LIN {X 0,Y 446.477,Z 468.872,A -85,B 0,C 180,E1 -8659.303,E2 -8659.303} C_VEL
LIN {X 0,Y 446.426,Z 468.876,A -85,B 0,C 180,E1 -8662.2,E2 -8662.2} C_VEL
LIN {X 0,Y 446.445,Z 468.875,A -85,B 0,C 180,E1 -8665.153,E2 -8665.153} C_VEL
LIN {X 0,Y 446.494,Z 468.867,A -85,B 0,C 180,E1 -8668.178,E2 -8668.178} C_VEL
LIN {X 0,Y 446.427,Z 468.873,A -85,B 0,C 180,E1 -8671.774,E2 -8671.774} C_VEL
LIN {X 0,Y 446.437,Z 468.875,A -85,B 0,C 180,E1 -8674.523,E2 -8674.523} C_VEL
LIN {X 0,Y 446.423,Z 468.875,A -85,B 0,C 180,E1 -8678.079,E2 -8678.079} C_VEL
LIN {X 0,Y 446.435,Z 468.877,A -85,B 0,C 180,E1 -8680.917,E2 -8680.917} C_VEL
LIN {X 0,Y 446.408,Z 468.878,A -85,B 0,C 180,E1 -8683.846,E2 -8683.846} C_VEL
LIN {X 0,Y 446.406,Z 468.879,A -85,B 0,C 180,E1 -8686.403,E2 -8686.403} C_VEL
LIN {X 0,Y 446.435,Z 468.875,A -85,B 0,C 180,E1 -8689.082,E2 -8689.082} C_VEL
LIN {X 0,Y 446.412,Z 468.861,A -85,B 0,C 180,E1 -8692.12,E2 -8692.12} C_VEL
LIN {X 0,Y 446.428,Z 468.864,A -85,B 0,C 180,E1 -8695.475,E2 -8695.475} C_VEL
LIN {X 0,Y 446.475,Z 469.066,A -85,B 0,C 180,E1 -8698.572,E2 -8698.572} C_VEL
LIN {X 0,Y 449.548,Z 481.832,A -85,B 0,C 180,E1 -8700.754,E2 -8700.754} C_VEL
LIN {X 0,Y 450.889,Z 488.731,A -85,B 0,C 180,E1 -8701.866,E2 -8701.866} C_VEL
LIN {X 0,Y 450.438,Z 498.912,A -85,B 0,C 180,E1 -8703.346,E2 -8703.346} C_VEL
LIN {X 0,Y 449.183,Z 522.67,A -85,B 0,C 180,E1 -8706.728,E2 -8706.728} C_VEL
LIN {X 0,Y 447.86,Z 550.31,A -85,B 0,C 180,E1 -8710.583,E2 -8710.583} C_VEL
LIN {X 0,Y 447.484,Z 560.999,A -85,B 0,C 180,E1 -8712.017,E2 -8712.017} C_VEL
LIN {X 0,Y 450.722,Z 590.947,A -85,B 0,C 180,E1 -8712.672,E2 -8712.672} C_VEL
LIN {X 0,Y 449.9,Z 671.631,A -85,B 0,C 180,E1 -8713.988,E2 -8713.988} C_VEL
LIN {X 0,Y 449.488,Z 684.888,A -85,B 0,C 180,E1 -8714.38,E2 -8714.38} C_VEL
LIN {X 0,Y 448.906,Z 697.096,A -85,B 0,C 180,E1 -8714.912,E2 -8714.912} C_VEL
LIN {X 0,Y 448.274,Z 708.646,A -85,B 0,C 180,E1 -8715.587,E2 -8715.587} C_VEL
LIN {X 0,Y 447.599,Z 720.331,A -85,B 0,C 180,E1 -8716.472,E2 -8716.472} C_VEL
LIN {X 0,Y 447.145,Z 732.388,A -85,B 0,C 180,E1 -8717.518,E2 -8717.518} C_VEL
LIN {X 0,Y 446.594,Z 740.995,A -85,B 0,C 180,E1 -8718.424,E2 -8718.424} C_VEL
LIN {X 0,Y 446.277,Z 749.935,A -85,B 0,C 180,E1 -8719.565,E2 -8719.565} C_VEL
LIN {X 0,Y 445.963,Z 758.561,A -85,B 0,C 180,E1 -8720.931,E2 -8720.931} C_VEL
LIN {X 0,Y 445.725,Z 765.492,A -85,B 0,C 180,E1 -8722.296,E2 -8722.296} C_VEL
LIN {X 0,Y 445.62,Z 771.01,A -85,B 0,C 180,E1 -8723.66,E2 -8723.66} C_VEL
LIN {X 0,Y 445.591,Z 775.282,A -85,B 0,C 180,E1 -8725.022,E2 -8725.022} C_VEL
LIN {X 0,Y 445.584,Z 778.435,A -85,B 0,C 180,E1 -8726.381,E2 -8726.381} C_VEL
LIN {X 0,Y 445.572,Z 779.958,A -85,B 0,C 180,E1 -8727.286,E2 -8727.286} C_VEL
LIN {X 0,Y 445.593,Z 781.035,A -85,B 0,C 180,E1 -8728.191,E2 -8728.191} C_VEL
LIN {X 0,Y 445.531,Z 781.699,A -85,B 0,C 180,E1 -8729.095,E2 -8729.095} C_VEL
LIN {X 0,Y 445.555,Z 781.947,A -85,B 0,C 180,E1 -8729.998,E2 -8729.998} C_VEL
LIN {X 0,Y 445.528,Z 781.728,A -85,B 0,C 180,E1 -8730.902,E2 -8730.902} C_VEL
LIN {X 0,Y 445.589,Z 781.104,A -85,B 0,C 180,E1 -8731.806,E2 -8731.806} C_VEL
LIN {X 0,Y 445.567,Z 780.065,A -85,B 0,C 180,E1 -8732.711,E2 -8732.711} C_VEL
LIN {X 0,Y 445.573,Z 778.556,A -85,B 0,C 180,E1 -8733.616,E2 -8733.616} C_VEL
LIN {X 0,Y 445.578,Z 775.446,A -85,B 0,C 180,E1 -8734.975,E2 -8734.975} C_VEL
LIN {X 0,Y 445.604,Z 770.735,A -85,B 0,C 180,E1 -8736.47,E2 -8736.47} C_VEL
LIN {X 0,Y 445.745,Z 764.718,A -85,B 0,C 180,E1 -8737.928,E2 -8737.928} C_VEL
LIN {X 0,Y 445.979,Z 757.563,A -85,B 0,C 180,E1 -8739.294,E2 -8739.294} C_VEL
LIN {X 0,Y 446.321,Z 748.559,A -85,B 0,C 180,E1 -8740.661,E2 -8740.661} C_VEL
LIN {X 0,Y 446.658,Z 739.29,A -85,B 0,C 180,E1 -8741.802,E2 -8741.802} C_VEL
LIN {X 0,Y 447.233,Z 730.265,A -85,B 0,C 180,E1 -8742.707,E2 -8742.707} C_VEL
LIN {X 0,Y 447.641,Z 719.058,A -85,B 0,C 180,E1 -8743.619,E2 -8743.619} C_VEL
LIN {X 0,Y 448.409,Z 703.786,A -85,B 0,C 180,E1 -8744.637,E2 -8744.637} C_VEL
LIN {X 0,Y 448.973,Z 691.565,A -85,B 0,C 180,E1 -8745.257,E2 -8745.257} C_VEL
LIN {X 0,Y 449.538,Z 678.317,A -85,B 0,C 180,E1 -8745.731,E2 -8745.731} C_VEL
LIN {X 0,Y 449.81,Z 665.485,A -85,B 0,C 180,E1 -8746.012,E2 -8746.012} C_VEL
LIN {X 0,Y 450.296,Z 588.926,A -85,B 0,C 180,E1 -8747.238,E2 -8747.238} C_VEL
LIN {X 0,Y 447.405,Z 561.671,A -85,B 0,C 180,E1 -8747.804,E2 -8747.804} C_VEL
LIN {X 0,Y 448.284,Z 537.227,A -85,B 0,C 180,E1 -8751.134,E2 -8751.134} C_VEL
LIN {X 0,Y 449.315,Z 514.727,A -85,B 0,C 180,E1 -8754.24,E2 -8754.24} C_VEL
LIN {X 0,Y 450.483,Z 491.581,A -85,B 0,C 180,E1 -8757.481,E2 -8757.481} C_VEL
LIN {X 0,Y 450.402,Z 486.851,A -85,B 0,C 180,E1 -8758.163,E2 -8758.163} C_VEL
LIN {X 0,Y 446.49,Z 468.988,A -85,B 0,C 180,E1 -8760.996,E2 -8760.996} C_VEL
LIN {X 0,Y 446.416,Z 468.879,A -85,B 0,C 180,E1 -8764.522,E2 -8764.522} C_VEL
LIN {X 0,Y 446.392,Z 468.883,A -85,B 0,C 180,E1 -8768.075,E2 -8768.075} C_VEL
LIN {X 0,Y 446.398,Z 468.875,A -85,B 0,C 180,E1 -8771.392,E2 -8771.392} C_VEL
LIN {X 0,Y 446.441,Z 468.87,A -85,B 0,C 180,E1 -8775.102,E2 -8775.102} C_VEL
LIN {X 0,Y 446.401,Z 468.878,A -85,B 0,C 180,E1 -8778.605,E2 -8778.605} C_VEL
LIN {X 0,Y 446.4,Z 468.878,A -85,B 0,C 180,E1 -8781.92,E2 -8781.92} C_VEL
LIN {X 0,Y 446.417,Z 468.873,A -85,B 0,C 180,E1 -8785.476,E2 -8785.476} C_VEL
LIN {X 0,Y 446.404,Z 468.877,A -85,B 0,C 180,E1 -8788.698,E2 -8788.698} C_VEL
LIN {X 0,Y 446.473,Z 468.867,A -85,B 0,C 180,E1 -8791.82,E2 -8791.82} C_VEL
LIN {X 0,Y 446.426,Z 468.874,A -85,B 0,C 180,E1 -8794.845,E2 -8794.845} C_VEL
LIN {X 0,Y 446.435,Z 468.876,A -85,B 0,C 180,E1 -8798.244,E2 -8798.244} C_VEL
LIN {X 0,Y 446.442,Z 468.87,A -85,B 0,C 180,E1 -8801.648,E2 -8801.648} C_VEL
LIN {X 0,Y 446.493,Z 468.871,A -85,B 0,C 180,E1 -8804.479,E2 -8804.479} C_VEL
LIN {X 0,Y 446.505,Z 468.866,A -85,B 0,C 180,E1 -8808.192,E2 -8808.192} C_VEL
LIN {X 0,Y 446.586,Z 468.853,A -85,B 0,C 180,E1 -8811.857,E2 -8811.857} C_VEL
LIN {X 0,Y 446.624,Z 468.854,A -85,B 0,C 180,E1 -8814.582,E2 -8814.582} C_VEL
LIN {X 0,Y 446.651,Z 468.847,A -85,B 0,C 180,E1 -8818.196,E2 -8818.196} C_VEL
LIN {X 0,Y 446.778,Z 468.829,A -85,B 0,C 180,E1 -8820,E2 -8820} C_VEL
LIN {X 0,Y 446.694,Z 468.844,A -85,B 0,C 180,E1 -8822.705,E2 -8822.705} C_VEL
LIN {X 0,Y 446.624,Z 468.851,A -85,B 0,C 180,E1 -8826.324,E2 -8826.324} C_VEL
LIN {X 0,Y 446.525,Z 468.862,A -85,B 0,C 180,E1 -8829.055,E2 -8829.055} C_VEL
LIN {X 0,Y 446.507,Z 468.868,A -85,B 0,C 180,E1 -8832.73,E2 -8832.73} C_VEL
LIN {X 0,Y 446.482,Z 468.867,A -85,B 0,C 180,E1 -8836.228,E2 -8836.228} C_VEL
LIN {X 0,Y 446.455,Z 468.869,A -85,B 0,C 180,E1 -8839.303,E2 -8839.303} C_VEL
LIN {X 0,Y 446.404,Z 468.876,A -85,B 0,C 180,E1 -8842.2,E2 -8842.2} C_VEL
LIN {X 0,Y 446.444,Z 468.872,A -85,B 0,C 180,E1 -8845.153,E2 -8845.153} C_VEL
LIN {X 0,Y 446.471,Z 468.867,A -85,B 0,C 180,E1 -8848.179,E2 -8848.179} C_VEL
LIN {X 0,Y 446.406,Z 468.874,A -85,B 0,C 180,E1 -8851.776,E2 -8851.776} C_VEL
LIN {X 0,Y 446.417,Z 468.877,A -85,B 0,C 180,E1 -8854.524,E2 -8854.524} C_VEL
LIN {X 0,Y 446.418,Z 468.873,A -85,B 0,C 180,E1 -8858.083,E2 -8858.083} C_VEL
LIN {X 0,Y 446.416,Z 468.88,A -85,B 0,C 180,E1 -8860.919,E2 -8860.919} C_VEL
LIN {X 0,Y 446.414,Z 468.873,A -85,B 0,C 180,E1 -8863.844,E2 -8863.844} C_VEL
LIN {X 0,Y 446.436,Z 468.872,A -85,B 0,C 180,E1 -8866.398,E2 -8866.398} C_VEL
LIN {X 0,Y 446.459,Z 468.867,A -85,B 0,C 180,E1 -8869.806,E2 -8869.806} C_VEL
LIN {X 0,Y 446.424,Z 468.872,A -85,B 0,C 180,E1 -8872.125,E2 -8872.125} C_VEL
LIN {X 0,Y 446.421,Z 468.874,A -85,B 0,C 180,E1 -8875.478,E2 -8875.478} C_VEL
LIN {X 0,Y 446.408,Z 468.878,A -85,B 0,C 180,E1 -8878.701,E2 -8878.701} C_VEL
LIN {X 0,Y 446.476,Z 468.865,A -85,B 0,C 180,E1 -8881.823,E2 -8881.823} C_VEL
LIN {X 0,Y 446.451,Z 468.874,A -85,B 0,C 180,E1 -8884.849,E2 -8884.849} C_VEL
LIN {X 0,Y 446.442,Z 468.87,A -85,B 0,C 180,E1 -8888.246,E2 -8888.246} C_VEL
LIN {X 0,Y 446.452,Z 468.87,A -85,B 0,C 180,E1 -8891.651,E2 -8891.651} C_VEL
LIN {X 0,Y 446.503,Z 468.863,A -85,B 0,C 180,E1 -8894.481,E2 -8894.481} C_VEL
LIN {X 0,Y 446.514,Z 468.86,A -85,B 0,C 180,E1 -8898.195,E2 -8898.195} C_VEL
LIN {X 0,Y 446.597,Z 468.855,A -85,B 0,C 180,E1 -8901.859,E2 -8901.859} C_VEL
LIN {X 0,Y 446.645,Z 468.85,A -85,B 0,C 180,E1 -8904.584,E2 -8904.584} C_VEL
LIN {X 0,Y 446.462,Z 468.873,A -85,B 0,C 180,E1 -8905.655,E2 -8905.655} C_VEL
LIN {X 0,Y 446.343,Z 469.733,A -85,B 0,C 180,E1 -8906.036,E2 -8906.036} C_VEL
LIN {X 0,Y 446,Z 472.43,A -85,B 0,C 180,E1 -8906.43,E2 -8906.43} C_VEL
LIN {X 0,Y 445.49,Z 476.63,A -85,B 0,C 180,E1 -8906.744,E2 -8906.744} C_VEL
LIN {X 0,Y 444.895,Z 481.645,A -85,B 0,C 180,E1 -8906.929,E2 -8906.929} C_VEL
LIN {X 0,Y 444.052,Z 488.483,A -85,B 0,C 180,E1 -8907.053,E2 -8907.053} C_VEL
LIN {X 0,Y 443.816,Z 497.703,A -85,B 0,C 180,E1 -8907.197,E2 -8907.197} C_VEL
LIN {X 0,Y 443.446,Z 550.424,A -85,B 0,C 180,E1 -8908.072,E2 -8908.072} C_VEL
LIN {X 0,Y 443.362,Z 563.699,A -85,B 0,C 180,E1 -8908.469,E2 -8908.469} C_VEL
LIN {X 0,Y 443.164,Z 576.191,A -85,B 0,C 180,E1 -8909.029,E2 -8909.029} C_VEL
LIN {X 0,Y 442.841,Z 588.103,A -85,B 0,C 180,E1 -8909.752,E2 -8909.752} C_VEL
LIN {X 0,Y 442.363,Z 599.846,A -85,B 0,C 180,E1 -8910.684,E2 -8910.684} C_VEL
LIN {X 0,Y 441.805,Z 610.165,A -85,B 0,C 180,E1 -8911.711,E2 -8911.711} C_VEL
LIN {X 0,Y 441.426,Z 618.569,A -85,B 0,C 180,E1 -8912.739,E2 -8912.739} C_VEL
LIN {X 0,Y 440.972,Z 626.354,A -85,B 0,C 180,E1 -8913.885,E2 -8913.885} C_VEL
LIN {X 0,Y 440.548,Z 633.965,A -85,B 0,C 180,E1 -8915.265,E2 -8915.265} C_VEL
LIN {X 0,Y 440.134,Z 640.974,A -85,B 0,C 180,E1 -8916.88,E2 -8916.88} C_VEL
LIN {X 0,Y 439.824,Z 645.658,A -85,B 0,C 180,E1 -8918.27,E2 -8918.27} C_VEL
LIN {X 0,Y 439.587,Z 649.245,A -85,B 0,C 180,E1 -8919.666,E2 -8919.666} C_VEL
LIN {X 0,Y 439.392,Z 651.829,A -85,B 0,C 180,E1 -8921.067,E2 -8921.067} C_VEL
LIN {X 0,Y 439.334,Z 653.59,A -85,B 0,C 180,E1 -8922.629,E2 -8922.629} C_VEL
LIN {X 0,Y 439.316,Z 654.165,A -85,B 0,C 180,E1 -8923.886,E2 -8923.886} C_VEL
LIN {X 0,Y 439.329,Z 654.148,A -85,B 0,C 180,E1 -8924.832,E2 -8924.832} C_VEL
LIN {X 0,Y 439.453,Z 653.235,A -85,B 0,C 180,E1 -8926.352,E2 -8926.352} C_VEL
LIN {X 0,Y 439.592,Z 651.532,A -85,B 0,C 180,E1 -8927.685,E2 -8927.685} C_VEL
LIN {X 0,Y 439.838,Z 648.839,A -85,B 0,C 180,E1 -8929.076,E2 -8929.076} C_VEL
LIN {X 0,Y 440.172,Z 644.841,A -85,B 0,C 180,E1 -8930.566,E2 -8930.566} C_VEL
LIN {X 0,Y 440.575,Z 640.008,A -85,B 0,C 180,E1 -8931.938,E2 -8931.938} C_VEL
LIN {X 0,Y 441.03,Z 634.312,A -85,B 0,C 180,E1 -8933.23,E2 -8933.23} C_VEL
LIN {X 0,Y 441.595,Z 626.745,A -85,B 0,C 180,E1 -8934.612,E2 -8934.612} C_VEL
LIN {X 0,Y 442.19,Z 617.836,A -85,B 0,C 180,E1 -8935.919,E2 -8935.919} C_VEL
LIN {X 0,Y 442.747,Z 608.82,A -85,B 0,C 180,E1 -8936.995,E2 -8936.995} C_VEL
LIN {X 0,Y 443.35,Z 598.313,A -85,B 0,C 180,E1 -8938.011,E2 -8938.011} C_VEL
LIN {X 0,Y 443.885,Z 586.926,A -85,B 0,C 180,E1 -8938.877,E2 -8938.877} C_VEL
LIN {X 0,Y 444.236,Z 574.989,A -85,B 0,C 180,E1 -8939.581,E2 -8939.581} C_VEL
LIN {X 0,Y 444.407,Z 562.171,A -85,B 0,C 180,E1 -8940.133,E2 -8940.133} C_VEL
LIN {X 0,Y 444.504,Z 548.688,A -85,B 0,C 180,E1 -8940.496,E2 -8940.496} C_VEL
LIN {X 0,Y 445.006,Z 483.958,A -85,B 0,C 180,E1 -8941.582,E2 -8941.582} C_VEL
LIN {X 0,Y 439.597,Z 470.681,A -85,B 0,C 180,E1 -8942.108,E2 -8942.108} C_VEL
LIN {X 0,Y 439.42,Z 469.824,A -85,B 0,C 180,E1 -8942.299,E2 -8942.299} C_VEL
LIN {X 0,Y 439.395,Z 469.751,A -85,B 0,C 180,E1 -8945.341,E2 -8945.341} C_VEL
LIN {X 0,Y 439.379,Z 469.757,A -85,B 0,C 180,E1 -8948.597,E2 -8948.597} C_VEL
LIN {X 0,Y 439.393,Z 469.752,A -85,B 0,C 180,E1 -8951.258,E2 -8951.258} C_VEL
LIN {X 0,Y 439.404,Z 469.753,A -85,B 0,C 180,E1 -8954.731,E2 -8954.731} C_VEL
LIN {X 0,Y 439.401,Z 469.752,A -85,B 0,C 180,E1 -8957.797,E2 -8957.797} C_VEL
LIN {X 0,Y 439.449,Z 469.899,A -85,B 0,C 180,E1 -8960.531,E2 -8960.531} C_VEL
LIN {X 0,Y 442.432,Z 484.435,A -85,B 0,C 180,E1 -8963.155,E2 -8963.155} C_VEL
LIN {X 0,Y 441.997,Z 500.844,A -85,B 0,C 180,E1 -8965.883,E2 -8965.883} C_VEL
LIN {X 0,Y 441.36,Z 520.086,A -85,B 0,C 180,E1 -8969.045,E2 -8969.045} C_VEL
LIN {X 0,Y 442.817,Z 528.551,A -85,B 0,C 180,E1 -8969.296,E2 -8969.296} C_VEL
LIN {X 0,Y 444.048,Z 537.306,A -85,B 0,C 180,E1 -8969.507,E2 -8969.507} C_VEL
LIN {X 0,Y 442.745,Z 630.209,A -85,B 0,C 180,E1 -8971.187,E2 -8971.187} C_VEL
LIN {X 0,Y 442.439,Z 643.262,A -85,B 0,C 180,E1 -8971.605,E2 -8971.605} C_VEL
LIN {X 0,Y 441.965,Z 656.195,A -85,B 0,C 180,E1 -8972.218,E2 -8972.218} C_VEL
LIN {X 0,Y 441.538,Z 668.066,A -85,B 0,C 180,E1 -8972.97,E2 -8972.97} C_VEL
LIN {X 0,Y 440.979,Z 679.22,A -85,B 0,C 180,E1 -8973.879,E2 -8973.879} C_VEL
LIN {X 0,Y 440.37,Z 690.05,A -85,B 0,C 180,E1 -8974.981,E2 -8974.981} C_VEL
LIN {X 0,Y 439.881,Z 699.698,A -85,B 0,C 180,E1 -8976.208,E2 -8976.208} C_VEL
LIN {X 0,Y 439.385,Z 708.731,A -85,B 0,C 180,E1 -8977.635,E2 -8977.635} C_VEL
LIN {X 0,Y 438.971,Z 716.196,A -85,B 0,C 180,E1 -8979.132,E2 -8979.132} C_VEL
LIN {X 0,Y 438.729,Z 722.312,A -85,B 0,C 180,E1 -8980.705,E2 -8980.705} C_VEL
LIN {X 0,Y 438.498,Z 726.876,A -85,B 0,C 180,E1 -8982.271,E2 -8982.271} C_VEL
LIN {X 0,Y 438.419,Z 728.978,A -85,B 0,C 180,E1 -8983.229,E2 -8983.229} C_VEL
LIN {X 0,Y 438.327,Z 730.625,A -85,B 0,C 180,E1 -8984.183,E2 -8984.183} C_VEL
LIN {X 0,Y 438.293,Z 731.781,A -85,B 0,C 180,E1 -8985.134,E2 -8985.134} C_VEL
LIN {X 0,Y 438.252,Z 732.499,A -85,B 0,C 180,E1 -8986.082,E2 -8986.082} C_VEL
LIN {X 0,Y 438.272,Z 732.802,A -85,B 0,C 180,E1 -8987.027,E2 -8987.027} C_VEL
LIN {X 0,Y 438.381,Z 732.633,A -85,B 0,C 180,E1 -8987.971,E2 -8987.971} C_VEL
LIN {X 0,Y 438.381,Z 732.047,A -85,B 0,C 180,E1 -8988.909,E2 -8988.909} C_VEL
LIN {X 0,Y 438.369,Z 731.061,A -85,B 0,C 180,E1 -8989.843,E2 -8989.843} C_VEL
LIN {X 0,Y 438.443,Z 729.611,A -85,B 0,C 180,E1 -8990.776,E2 -8990.776} C_VEL
LIN {X 0,Y 438.654,Z 726.595,A -85,B 0,C 180,E1 -8992.173,E2 -8992.173} C_VEL
LIN {X 0,Y 438.836,Z 722.512,A -85,B 0,C 180,E1 -8993.564,E2 -8993.564} C_VEL
LIN {X 0,Y 439.121,Z 716.276,A -85,B 0,C 180,E1 -8995.18,E2 -8995.18} C_VEL
LIN {X 0,Y 439.472,Z 709.438,A -85,B 0,C 180,E1 -8996.562,E2 -8996.562} C_VEL
LIN {X 0,Y 440.004,Z 700.882,A -85,B 0,C 180,E1 -8997.941,E2 -8997.941} C_VEL
LIN {X 0,Y 440.58,Z 691.174,A -85,B 0,C 180,E1 -8999.201,E2 -8999.201} C_VEL
LIN {X 0,Y 441.227,Z 680.069,A -85,B 0,C 180,E1 -9000.343,E2 -9000.343} C_VEL
LIN {X 0,Y 441.8,Z 668.964,A -85,B 0,C 180,E1 -9001.254,E2 -9001.254} C_VEL
LIN {X 0,Y 442.291,Z 657.378,A -85,B 0,C 180,E1 -9001.992,E2 -9001.992} C_VEL
LIN {X 0,Y 442.762,Z 644.338,A -85,B 0,C 180,E1 -9002.616,E2 -9002.616} C_VEL
LIN {X 0,Y 443.053,Z 631.125,A -85,B 0,C 180,E1 -9003.041,E2 -9003.041} C_VEL
LIN {X 0,Y 444.582,Z 535.636,A -85,B 0,C 180,E1 -9004.853,E2 -9004.853} C_VEL
LIN {X 0,Y 442.01,Z 521.914,A -85,B 0,C 180,E1 -9005.295,E2 -9005.295} C_VEL
LIN {X 0,Y 442.645,Z 499.692,A -85,B 0,C 180,E1 -9008.906,E2 -9008.906} C_VEL
LIN {X 0,Y 443.011,Z 486.705,A -85,B 0,C 180,E1 -9010.975,E2 -9010.975} C_VEL
LIN {X 0,Y 441.276,Z 477.085,A -85,B 0,C 180,E1 -9012.65,E2 -9012.65} C_VEL
LIN {X 0,Y 439.441,Z 469.873,A -85,B 0,C 180,E1 -9013.969,E2 -9013.969} C_VEL
LIN {X 0,Y 439.456,Z 469.747,A -85,B 0,C 180,E1 -9016.731,E2 -9016.731} C_VEL
LIN {X 0,Y 439.41,Z 469.751,A -85,B 0,C 180,E1 -9019.626,E2 -9019.626} C_VEL
LIN {X 0,Y 439.372,Z 469.756,A -85,B 0,C 180,E1 -9022.575,E2 -9022.575} C_VEL
LIN {X 0,Y 439.394,Z 469.752,A -85,B 0,C 180,E1 -9025.586,E2 -9025.586} C_VEL
LIN {X 0,Y 439.426,Z 469.749,A -85,B 0,C 180,E1 -9028.673,E2 -9028.673} C_VEL
LIN {X 0,Y 439.378,Z 469.752,A -85,B 0,C 180,E1 -9032.03,E2 -9032.03} C_VEL
LIN {X 0,Y 439.403,Z 469.749,A -85,B 0,C 180,E1 -9035.34,E2 -9035.34} C_VEL
LIN {X 0,Y 439.386,Z 469.754,A -85,B 0,C 180,E1 -9038.595,E2 -9038.595} C_VEL
LIN {X 0,Y 439.397,Z 469.751,A -85,B 0,C 180,E1 -9041.256,E2 -9041.256} C_VEL
LIN {X 0,Y 439.408,Z 469.751,A -85,B 0,C 180,E1 -9044.729,E2 -9044.729} C_VEL
LIN {X 0,Y 439.404,Z 469.751,A -85,B 0,C 180,E1 -9047.795,E2 -9047.795} C_VEL
LIN {X 0,Y 439.397,Z 469.747,A -85,B 0,C 180,E1 -9050.223,E2 -9050.223} C_VEL
LIN {X 0,Y 439.379,Z 469.754,A -85,B 0,C 180,E1 -9053.712,E2 -9053.712} C_VEL
LIN {X 0,Y 439.378,Z 469.754,A -85,B 0,C 180,E1 -9057.053,E2 -9057.053} C_VEL
LIN {X 0,Y 439.408,Z 469.966,A -85,B 0,C 180,E1 -9058.242,E2 -9058.242} C_VEL
LIN {X 0,Y 442.211,Z 481.198,A -85,B 0,C 180,E1 -9060.22,E2 -9060.22} C_VEL
LIN {X 0,Y 443.966,Z 489.822,A -85,B 0,C 180,E1 -9061.646,E2 -9061.646} C_VEL
LIN {X 0,Y 444.057,Z 493.291,A -85,B 0,C 180,E1 -9062.178,E2 -9062.178} C_VEL
LIN {X 0,Y 442.567,Z 516.885,A -85,B 0,C 180,E1 -9065.613,E2 -9065.613} C_VEL
LIN {X 0,Y 441.379,Z 538.889,A -85,B 0,C 180,E1 -9068.761,E2 -9068.761} C_VEL
LIN {X 0,Y 440.535,Z 559.742,A -85,B 0,C 180,E1 -9071.674,E2 -9071.674} C_VEL
LIN {X 0,Y 443.258,Z 584.816,A -85,B 0,C 180,E1 -9072.251,E2 -9072.251} C_VEL
LIN {X 0,Y 443.978,Z 592.474,A -85,B 0,C 180,E1 -9072.412,E2 -9072.412} C_VEL
LIN {X 0,Y 443.12,Z 670.409,A -85,B 0,C 180,E1 -9073.707,E2 -9073.707} C_VEL
LIN {X 0,Y 442.711,Z 683.725,A -85,B 0,C 180,E1 -9074.106,E2 -9074.106} C_VEL
LIN {X 0,Y 442.024,Z 696.533,A -85,B 0,C 180,E1 -9074.671,E2 -9074.671} C_VEL
LIN {X 0,Y 441.371,Z 707.968,A -85,B 0,C 180,E1 -9075.357,E2 -9075.357} C_VEL
LIN {X 0,Y 440.365,Z 725.352,A -85,B 0,C 180,E1 -9076.701,E2 -9076.701} C_VEL
LIN {X 0,Y 439.949,Z 735.393,A -85,B 0,C 180,E1 -9077.662,E2 -9077.662} C_VEL
LIN {X 0,Y 439.51,Z 744.355,A -85,B 0,C 180,E1 -9078.702,E2 -9078.702} C_VEL
LIN {X 0,Y 439.078,Z 752.595,A -85,B 0,C 180,E1 -9079.858,E2 -9079.858} C_VEL
LIN {X 0,Y 438.812,Z 760.649,A -85,B 0,C 180,E1 -9081.247,E2 -9081.247} C_VEL
LIN {X 0,Y 438.614,Z 767.072,A -85,B 0,C 180,E1 -9082.634,E2 -9082.634} C_VEL
LIN {X 0,Y 438.496,Z 772.591,A -85,B 0,C 180,E1 -9084.154,E2 -9084.154} C_VEL
LIN {X 0,Y 438.47,Z 776.04,A -85,B 0,C 180,E1 -9085.402,E2 -9085.402} C_VEL
LIN {X 0,Y 438.48,Z 778.049,A -85,B 0,C 180,E1 -9086.323,E2 -9086.323} C_VEL
LIN {X 0,Y 438.495,Z 779.568,A -85,B 0,C 180,E1 -9087.242,E2 -9087.242} C_VEL
LIN {X 0,Y 438.5,Z 780.643,A -85,B 0,C 180,E1 -9088.162,E2 -9088.162} C_VEL
LIN {X 0,Y 438.465,Z 781.308,A -85,B 0,C 180,E1 -9089.08,E2 -9089.08} C_VEL
LIN {X 0,Y 438.484,Z 781.546,A -85,B 0,C 180,E1 -9089.998,E2 -9089.998} C_VEL
LIN {X 0,Y 438.462,Z 781.32,A -85,B 0,C 180,E1 -9090.917,E2 -9090.917} C_VEL
LIN {X 0,Y 438.496,Z 780.688,A -85,B 0,C 180,E1 -9091.835,E2 -9091.835} C_VEL
LIN {X 0,Y 438.489,Z 779.642,A -85,B 0,C 180,E1 -9092.754,E2 -9092.754} C_VEL
LIN {X 0,Y 438.472,Z 778.114,A -85,B 0,C 180,E1 -9093.674,E2 -9093.674} C_VEL
LIN {X 0,Y 438.507,Z 774.981,A -85,B 0,C 180,E1 -9095.056,E2 -9095.056} C_VEL
LIN {X 0,Y 438.505,Z 770.719,A -85,B 0,C 180,E1 -9096.44,E2 -9096.44} C_VEL
LIN {X 0,Y 438.688,Z 764.185,A -85,B 0,C 180,E1 -9098.057,E2 -9098.057} C_VEL
LIN {X 0,Y 438.911,Z 756.97,A -85,B 0,C 180,E1 -9099.445,E2 -9099.445} C_VEL
LIN {X 0,Y 439.31,Z 747.921,A -85,B 0,C 180,E1 -9100.833,E2 -9100.833} C_VEL
LIN {X 0,Y 439.641,Z 738.578,A -85,B 0,C 180,E1 -9101.993,E2 -9101.993} C_VEL
LIN {X 0,Y 440.218,Z 729.467,A -85,B 0,C 180,E1 -9102.913,E2 -9102.913} C_VEL
LIN {X 0,Y 440.662,Z 718.157,A -85,B 0,C 180,E1 -9103.839,E2 -9103.839} C_VEL
LIN {X 0,Y 441.63,Z 700.367,A -85,B 0,C 180,E1 -9104.985,E2 -9104.985} C_VEL
LIN {X 0,Y 442.234,Z 687.379,A -85,B 0,C 180,E1 -9105.613,E2 -9105.613} C_VEL
LIN {X 0,Y 442.72,Z 674.287,A -85,B 0,C 180,E1 -9106.039,E2 -9106.039} C_VEL
LIN {X 0,Y 443.012,Z 655.783,A -85,B 0,C 180,E1 -9106.383,E2 -9106.383} C_VEL
LIN {X 0,Y 443.553,Z 590.85,A -85,B 0,C 180,E1 -9107.436,E2 -9107.436} C_VEL
LIN {X 0,Y 440.399,Z 560.897,A -85,B 0,C 180,E1 -9108.056,E2 -9108.056} C_VEL
LIN {X 0,Y 441.264,Z 537.756,A -85,B 0,C 180,E1 -9111.242,E2 -9111.242} C_VEL
LIN {X 0,Y 442.442,Z 513.843,A -85,B 0,C 180,E1 -9114.604,E2 -9114.604} C_VEL
LIN {X 0,Y 443.65,Z 490.977,A -85,B 0,C 180,E1 -9117.858,E2 -9117.858} C_VEL
LIN {X 0,Y 443.017,Z 486.063,A -85,B 0,C 180,E1 -9118.604,E2 -9118.604} C_VEL
LIN {X 0,Y 439.427,Z 469.862,A -85,B 0,C 180,E1 -9121.232,E2 -9121.232} C_VEL
LIN {X 0,Y 439.378,Z 469.758,A -85,B 0,C 180,E1 -9124.042,E2 -9124.042} C_VEL
LIN {X 0,Y 439.333,Z 469.756,A -85,B 0,C 180,E1 -9126.884,E2 -9126.884} C_VEL
LIN {X 0,Y 439.337,Z 469.758,A -85,B 0,C 180,E1 -9129.839,E2 -9129.839} C_VEL
LIN {X 0,Y 439.335,Z 469.758,A -85,B 0,C 180,E1 -9132.62,E2 -9132.62} C_VEL
LIN {X 0,Y 439.39,Z 469.748,A -85,B 0,C 180,E1 -9135.269,E2 -9135.269} C_VEL
LIN {X 0,Y 439.361,Z 469.754,A -85,B 0,C 180,E1 -9138.745,E2 -9138.745} C_VEL
LIN {X 0,Y 439.354,Z 469.753,A -85,B 0,C 180,E1 -9141.608,E2 -9141.608} C_VEL
LIN {X 0,Y 439.387,Z 469.75,A -85,B 0,C 180,E1 -9144.843,E2 -9144.843} C_VEL
LIN {X 0,Y 439.361,Z 469.757,A -85,B 0,C 180,E1 -9148.138,E2 -9148.138} C_VEL
LIN {X 0,Y 439.421,Z 469.745,A -85,B 0,C 180,E1 -9151.597,E2 -9151.597} C_VEL
LIN {X 0,Y 439.375,Z 469.757,A -85,B 0,C 180,E1 -9154.413,E2 -9154.413} C_VEL
LIN {X 0,Y 439.35,Z 469.753,A -85,B 0,C 180,E1 -9157.423,E2 -9157.423} C_VEL
LIN {X 0,Y 439.428,Z 469.748,A -85,B 0,C 180,E1 -9160.662,E2 -9160.662} C_VEL
LIN {X 0,Y 439.448,Z 469.746,A -85,B 0,C 180,E1 -9164.224,E2 -9164.224} C_VEL
LIN {X 0,Y 439.471,Z 469.74,A -85,B 0,C 180,E1 -9168.001,E2 -9168.001} C_VEL
LIN {X 0,Y 439.534,Z 469.73,A -85,B 0,C 180,E1 -9171.726,E2 -9171.726} C_VEL
LIN {X 0,Y 439.6,Z 469.73,A -85,B 0,C 180,E1 -9174.495,E2 -9174.495} C_VEL
LIN {X 0,Y 439.621,Z 469.722,A -85,B 0,C 180,E1 -9178.167,E2 -9178.167} C_VEL
LIN {X 0,Y 439.748,Z 469.705,A -85,B 0,C 180,E1 -9180,E2 -9180} C_VEL
LIN {X 0,Y 439.64,Z 469.722,A -85,B 0,C 180,E1 -9182.748,E2 -9182.748} C_VEL
LIN {X 0,Y 439.599,Z 469.728,A -85,B 0,C 180,E1 -9186.425,E2 -9186.425} C_VEL
LIN {X 0,Y 439.487,Z 469.737,A -85,B 0,C 180,E1 -9189.202,E2 -9189.202} C_VEL
LIN {X 0,Y 439.451,Z 469.744,A -85,B 0,C 180,E1 -9192.938,E2 -9192.938} C_VEL
LIN {X 0,Y 439.433,Z 469.746,A -85,B 0,C 180,E1 -9196.349,E2 -9196.349} C_VEL
LIN {X 0,Y 439.388,Z 469.748,A -85,B 0,C 180,E1 -9199.627,E2 -9199.627} C_VEL
LIN {X 0,Y 439.351,Z 469.759,A -85,B 0,C 180,E1 -9202.576,E2 -9202.576} C_VEL
LIN {X 0,Y 439.391,Z 469.748,A -85,B 0,C 180,E1 -9205.585,E2 -9205.585} C_VEL
LIN {X 0,Y 439.404,Z 469.753,A -85,B 0,C 180,E1 -9208.674,E2 -9208.674} C_VEL
LIN {X 0,Y 439.357,Z 469.752,A -85,B 0,C 180,E1 -9212.031,E2 -9212.031} C_VEL
LIN {X 0,Y 439.383,Z 469.751,A -85,B 0,C 180,E1 -9215.342,E2 -9215.342} C_VEL
LIN {X 0,Y 439.371,Z 469.755,A -85,B 0,C 180,E1 -9218.596,E2 -9218.596} C_VEL
LIN {X 0,Y 439.377,Z 469.752,A -85,B 0,C 180,E1 -9221.258,E2 -9221.258} C_VEL
LIN {X 0,Y 439.396,Z 469.753,A -85,B 0,C 180,E1 -9224.729,E2 -9224.729} C_VEL
LIN {X 0,Y 439.402,Z 469.746,A -85,B 0,C 180,E1 -9227.799,E2 -9227.799} C_VEL
LIN {X 0,Y 439.442,Z 469.742,A -85,B 0,C 180,E1 -9230.231,E2 -9230.231} C_VEL
LIN {X 0,Y 439.367,Z 469.751,A -85,B 0,C 180,E1 -9233.714,E2 -9233.714} C_VEL
LIN {X 0,Y 439.364,Z 469.758,A -85,B 0,C 180,E1 -9237.055,E2 -9237.055} C_VEL
LIN {X 0,Y 439.374,Z 469.75,A -85,B 0,C 180,E1 -9240.276,E2 -9240.276} C_VEL
LIN {X 0,Y 439.422,Z 469.747,A -85,B 0,C 180,E1 -9243.398,E2 -9243.398} C_VEL
LIN {X 0,Y 439.38,Z 469.75,A -85,B 0,C 180,E1 -9246.431,E2 -9246.431} C_VEL
LIN {X 0,Y 439.383,Z 469.752,A -85,B 0,C 180,E1 -9249.399,E2 -9249.399} C_VEL
LIN {X 0,Y 439.426,Z 469.744,A -85,B 0,C 180,E1 -9252.311,E2 -9252.311} C_VEL
LIN {X 0,Y 439.443,Z 469.749,A -85,B 0,C 180,E1 -9255.176,E2 -9255.176} C_VEL
LIN {X 0,Y 439.48,Z 469.737,A -85,B 0,C 180,E1 -9258.003,E2 -9258.003} C_VEL
LIN {X 0,Y 439.545,Z 469.734,A -85,B 0,C 180,E1 -9261.728,E2 -9261.728} C_VEL
LIN {X 0,Y 439.621,Z 469.725,A -85,B 0,C 180,E1 -9264.497,E2 -9264.497} C_VEL
LIN {X 0,Y 439.477,Z 469.927,A -85,B 0,C 180,E1 -9266.438,E2 -9266.438} C_VEL
LIN {X 0,Y 439.764,Z 471.003,A -85,B 0,C 180,E1 -9266.592,E2 -9266.592} C_VEL
LIN {X 0,Y 443.948,Z 482.631,A -85,B 0,C 180,E1 -9266.953,E2 -9266.953} C_VEL
LIN {X 0,Y 443.816,Z 497.703,A -85,B 0,C 180,E1 -9267.197,E2 -9267.197} C_VEL
LIN {X 0,Y 443.12,Z 503.549,A -85,B 0,C 180,E1 -9267.269,E2 -9267.269} C_VEL
LIN {X 0,Y 437.287,Z 522.517,A -85,B 0,C 180,E1 -9267.377,E2 -9267.377} C_VEL
LIN {X 0,Y 436.633,Z 528.362,A -85,B 0,C 180,E1 -9267.452,E2 -9267.452} C_VEL
LIN {X 0,Y 436.576,Z 553.241,A -85,B 0,C 180,E1 -9267.897,E2 -9267.897} C_VEL
LIN {X 0,Y 436.478,Z 566.473,A -85,B 0,C 180,E1 -9268.325,E2 -9268.325} C_VEL
LIN {X 0,Y 436.264,Z 578.709,A -85,B 0,C 180,E1 -9268.905,E2 -9268.905} C_VEL
LIN {X 0,Y 435.94,Z 589.882,A -85,B 0,C 180,E1 -9269.618,E2 -9269.618} C_VEL
LIN {X 0,Y 435.455,Z 601.621,A -85,B 0,C 180,E1 -9270.58,E2 -9270.58} C_VEL
LIN {X 0,Y 434.873,Z 611.805,A -85,B 0,C 180,E1 -9271.622,E2 -9271.622} C_VEL
LIN {X 0,Y 434.432,Z 620.921,A -85,B 0,C 180,E1 -9272.783,E2 -9272.783} C_VEL
LIN {X 0,Y 433.84,Z 629.806,A -85,B 0,C 180,E1 -9274.182,E2 -9274.182} C_VEL
LIN {X 0,Y 433.427,Z 636.955,A -85,B 0,C 180,E1 -9275.585,E2 -9275.585} C_VEL
LIN {X 0,Y 433.114,Z 642.677,A -85,B 0,C 180,E1 -9276.992,E2 -9276.992} C_VEL
LIN {X 0,Y 432.769,Z 647.209,A -85,B 0,C 180,E1 -9278.406,E2 -9278.406} C_VEL
LIN {X 0,Y 432.598,Z 649.598,A -85,B 0,C 180,E1 -9279.351,E2 -9279.351} C_VEL
LIN {X 0,Y 432.474,Z 651.558,A -85,B 0,C 180,E1 -9280.299,E2 -9280.299} C_VEL
LIN {X 0,Y 432.35,Z 653.111,A -85,B 0,C 180,E1 -9281.25,E2 -9281.25} C_VEL
LIN {X 0,Y 432.329,Z 654.656,A -85,B 0,C 180,E1 -9282.745,E2 -9282.745} C_VEL
LIN {X 0,Y 432.299,Z 655.192,A -85,B 0,C 180,E1 -9284.116,E2 -9284.116} C_VEL
LIN {X 0,Y 432.337,Z 655.081,A -85,B 0,C 180,E1 -9285.077,E2 -9285.077} C_VEL
LIN {X 0,Y 432.459,Z 654.156,A -85,B 0,C 180,E1 -9286.5,E2 -9286.5} C_VEL
LIN {X 0,Y 432.623,Z 652.222,A -85,B 0,C 180,E1 -9287.98,E2 -9287.98} C_VEL
LIN {X 0,Y 432.952,Z 648.636,A -85,B 0,C 180,E1 -9289.696,E2 -9289.696} C_VEL
LIN {X 0,Y 433.405,Z 643.579,A -85,B 0,C 180,E1 -9291.4,E2 -9291.4} C_VEL
LIN {X 0,Y 433.881,Z 637.791,A -85,B 0,C 180,E1 -9292.878,E2 -9292.878} C_VEL
LIN {X 0,Y 434.53,Z 630.38,A -85,B 0,C 180,E1 -9294.359,E2 -9294.359} C_VEL
LIN {X 0,Y 435.12,Z 622.41,A -85,B 0,C 180,E1 -9295.647,E2 -9295.647} C_VEL
LIN {X 0,Y 435.821,Z 613.295,A -85,B 0,C 180,E1 -9296.843,E2 -9296.843} C_VEL
LIN {X 0,Y 436.334,Z 603.926,A -85,B 0,C 180,E1 -9297.848,E2 -9297.848} C_VEL
LIN {X 0,Y 436.987,Z 592.133,A -85,B 0,C 180,E1 -9298.849,E2 -9298.849} C_VEL
LIN {X 0,Y 437.41,Z 581.062,A -85,B 0,C 180,E1 -9299.588,E2 -9299.588} C_VEL
LIN {X 0,Y 437.69,Z 568.474,A -85,B 0,C 180,E1 -9300.219,E2 -9300.219} C_VEL
LIN {X 0,Y 437.809,Z 556.155,A -85,B 0,C 180,E1 -9300.643,E2 -9300.643} C_VEL
LIN {X 0,Y 437.835,Z 537.38,A -85,B 0,C 180,E1 -9301.015,E2 -9301.015} C_VEL
LIN {X 0,Y 438.401,Z 485.702,A -85,B 0,C 180,E1 -9301.882,E2 -9301.882} C_VEL
LIN {X 0,Y 432.634,Z 471.813,A -85,B 0,C 180,E1 -9302.445,E2 -9302.445} C_VEL
LIN {X 0,Y 432.407,Z 470.938,A -85,B 0,C 180,E1 -9302.561,E2 -9302.561} C_VEL
LIN {X 0,Y 432.354,Z 470.629,A -85,B 0,C 180,E1 -9302.995,E2 -9302.995} C_VEL
LIN {X 0,Y 432.34,Z 470.631,A -85,B 0,C 180,E1 -9305.819,E2 -9305.819} C_VEL
LIN {X 0,Y 432.331,Z 470.627,A -85,B 0,C 180,E1 -9309.346,E2 -9309.346} C_VEL
LIN {X 0,Y 432.337,Z 470.628,A -85,B 0,C 180,E1 -9311.798,E2 -9311.798} C_VEL
LIN {X 0,Y 432.338,Z 470.632,A -85,B 0,C 180,E1 -9314.348,E2 -9314.348} C_VEL
LIN {X 0,Y 432.325,Z 470.635,A -85,B 0,C 180,E1 -9317.017,E2 -9317.017} C_VEL
LIN {X 0,Y 432.439,Z 470.805,A -85,B 0,C 180,E1 -9320.306,E2 -9320.306} C_VEL
LIN {X 0,Y 435.55,Z 485.948,A -85,B 0,C 180,E1 -9323.054,E2 -9323.054} C_VEL
LIN {X 0,Y 435.058,Z 502.665,A -85,B 0,C 180,E1 -9325.851,E2 -9325.851} C_VEL
LIN {X 0,Y 434.461,Z 520.598,A -85,B 0,C 180,E1 -9328.8,E2 -9328.8} C_VEL
LIN {X 0,Y 437.236,Z 537.224,A -85,B 0,C 180,E1 -9329.244,E2 -9329.244} C_VEL
LIN {X 0,Y 435.889,Z 630.079,A -85,B 0,C 180,E1 -9330.958,E2 -9330.958} C_VEL
LIN {X 0,Y 435.563,Z 643.223,A -85,B 0,C 180,E1 -9331.379,E2 -9331.379} C_VEL
LIN {X 0,Y 435.05,Z 656.231,A -85,B 0,C 180,E1 -9331.999,E2 -9331.999} C_VEL
LIN {X 0,Y 434.594,Z 668.718,A -85,B 0,C 180,E1 -9332.804,E2 -9332.804} C_VEL
LIN {X 0,Y 433.954,Z 680.73,A -85,B 0,C 180,E1 -9333.812,E2 -9333.812} C_VEL
LIN {X 0,Y 433.331,Z 691.347,A -85,B 0,C 180,E1 -9334.931,E2 -9334.931} C_VEL
LIN {X 0,Y 432.88,Z 699.962,A -85,B 0,C 180,E1 -9336.054,E2 -9336.054} C_VEL
LIN {X 0,Y 432.419,Z 707.97,A -85,B 0,C 180,E1 -9337.32,E2 -9337.32} C_VEL
LIN {X 0,Y 432.007,Z 715.45,A -85,B 0,C 180,E1 -9338.779,E2 -9338.779} C_VEL
LIN {X 0,Y 431.737,Z 720.515,A -85,B 0,C 180,E1 -9340.011,E2 -9340.011} C_VEL
LIN {X 0,Y 431.53,Z 725.325,A -85,B 0,C 180,E1 -9341.484,E2 -9341.484} C_VEL
LIN {X 0,Y 431.373,Z 728.884,A -85,B 0,C 180,E1 -9342.947,E2 -9342.947} C_VEL
LIN {X 0,Y 431.247,Z 730.854,A -85,B 0,C 180,E1 -9344.057,E2 -9344.057} C_VEL
LIN {X 0,Y 431.218,Z 731.939,A -85,B 0,C 180,E1 -9344.885,E2 -9344.885} C_VEL
LIN {X 0,Y 431.165,Z 732.762,A -85,B 0,C 180,E1 -9345.848,E2 -9345.848} C_VEL
LIN {X 0,Y 431.19,Z 733.152,A -85,B 0,C 180,E1 -9346.81,E2 -9346.81} C_VEL
LIN {X 0,Y 431.282,Z 733.092,A -85,B 0,C 180,E1 -9347.892,E2 -9347.892} C_VEL
LIN {X 0,Y 431.295,Z 731.741,A -85,B 0,C 180,E1 -9349.674,E2 -9349.674} C_VEL
LIN {X 0,Y 431.367,Z 730.427,A -85,B 0,C 180,E1 -9350.624,E2 -9350.624} C_VEL
LIN {X 0,Y 431.567,Z 727.591,A -85,B 0,C 180,E1 -9352.044,E2 -9352.044} C_VEL
LIN {X 0,Y 431.734,Z 723.711,A -85,B 0,C 180,E1 -9353.457,E2 -9353.457} C_VEL
LIN {X 0,Y 431.982,Z 718.655,A -85,B 0,C 180,E1 -9354.867,E2 -9354.867} C_VEL
LIN {X 0,Y 432.345,Z 712.266,A -85,B 0,C 180,E1 -9356.272,E2 -9356.272} C_VEL
LIN {X 0,Y 432.882,Z 704.316,A -85,B 0,C 180,E1 -9357.674,E2 -9357.674} C_VEL
LIN {X 0,Y 433.42,Z 696.204,A -85,B 0,C 180,E1 -9358.839,E2 -9358.839} C_VEL
LIN {X 0,Y 434.029,Z 686.229,A -85,B 0,C 180,E1 -9360,E2 -9360} C_VEL
LIN {X 0,Y 434.657,Z 675.107,A -85,B 0,C 180,E1 -9361.043,E2 -9361.043} C_VEL
LIN {X 0,Y 435.174,Z 664.267,A -85,B 0,C 180,E1 -9361.851,E2 -9361.851} C_VEL
LIN {X 0,Y 435.797,Z 651.025,A -85,B 0,C 180,E1 -9362.6,E2 -9362.6} C_VEL
LIN {X 0,Y 436.151,Z 638.326,A -85,B 0,C 180,E1 -9363.118,E2 -9363.118} C_VEL
LIN {X 0,Y 436.411,Z 624.995,A -85,B 0,C 180,E1 -9363.463,E2 -9363.463} C_VEL
LIN {X 0,Y 437.956,Z 536.823,A -85,B 0,C 180,E1 -9365.159,E2 -9365.159} C_VEL
LIN {X 0,Y 435.372,Z 523.29,A -85,B 0,C 180,E1 -9365.587,E2 -9365.587} C_VEL
LIN {X 0,Y 435.227,Z 522.142,A -85,B 0,C 180,E1 -9365.677,E2 -9365.677} C_VEL
LIN {X 0,Y 435.882,Z 500.126,A -85,B 0,C 180,E1 -9369.279,E2 -9369.279} C_VEL
LIN {X 0,Y 436.313,Z 488.638,A -85,B 0,C 180,E1 -9371.145,E2 -9371.145} C_VEL
LIN {X 0,Y 434.821,Z 480.226,A -85,B 0,C 180,E1 -9372.604,E2 -9372.604} C_VEL
LIN {X 0,Y 432.405,Z 470.769,A -85,B 0,C 180,E1 -9374.351,E2 -9374.351} C_VEL
LIN {X 0,Y 432.397,Z 470.626,A -85,B 0,C 180,E1 -9377.012,E2 -9377.012} C_VEL
LIN {X 0,Y 432.347,Z 470.63,A -85,B 0,C 180,E1 -9379.96,E2 -9379.96} C_VEL
LIN {X 0,Y 432.325,Z 470.636,A -85,B 0,C 180,E1 -9382.964,E2 -9382.964} C_VEL
LIN {X 0,Y 432.358,Z 470.628,A -85,B 0,C 180,E1 -9386.033,E2 -9386.033} C_VEL
LIN {X 0,Y 432.351,Z 470.631,A -85,B 0,C 180,E1 -9389.187,E2 -9389.187} C_VEL
LIN {X 0,Y 432.332,Z 470.631,A -85,B 0,C 180,E1 -9392.443,E2 -9392.443} C_VEL
LIN {X 0,Y 432.353,Z 470.627,A -85,B 0,C 180,E1 -9395.631,E2 -9395.631} C_VEL
LIN {X 0,Y 432.349,Z 470.631,A -85,B 0,C 180,E1 -9398.714,E2 -9398.714} C_VEL
LIN {X 0,Y 432.342,Z 470.63,A -85,B 0,C 180,E1 -9401.797,E2 -9401.797} C_VEL
LIN {X 0,Y 432.342,Z 470.63,A -85,B 0,C 180,E1 -9404.347,E2 -9404.347} C_VEL
LIN {X 0,Y 432.328,Z 470.633,A -85,B 0,C 180,E1 -9407.015,E2 -9407.015} C_VEL
LIN {X 0,Y 432.342,Z 470.632,A -85,B 0,C 180,E1 -9409.82,E2 -9409.82} C_VEL
LIN {X 0,Y 432.311,Z 470.627,A -85,B 0,C 180,E1 -9413.021,E2 -9413.021} C_VEL
LIN {X 0,Y 432.34,Z 470.617,A -85,B 0,C 180,E1 -9416.001,E2 -9416.001} C_VEL
LIN {X 0,Y 432.373,Z 470.87,A -85,B 0,C 180,E1 -9417.904,E2 -9417.904} C_VEL
LIN {X 0,Y 435.499,Z 483.434,A -85,B 0,C 180,E1 -9420.155,E2 -9420.155} C_VEL
LIN {X 0,Y 437.246,Z 492.624,A -85,B 0,C 180,E1 -9421.694,E2 -9421.694} C_VEL
LIN {X 0,Y 435.956,Z 513.687,A -85,B 0,C 180,E1 -9424.837,E2 -9424.837} C_VEL
LIN {X 0,Y 434.589,Z 536.473,A -85,B 0,C 180,E1 -9428.163,E2 -9428.163} C_VEL
LIN {X 0,Y 433.593,Z 558.386,A -85,B 0,C 180,E1 -9431.302,E2 -9431.302} C_VEL
LIN {X 0,Y 433.902,Z 561.281,A -85,B 0,C 180,E1 -9431.417,E2 -9431.417} C_VEL
LIN {X 0,Y 437.259,Z 592.031,A -85,B 0,C 180,E1 -9432.108,E2 -9432.108} C_VEL
LIN {X 0,Y 436.358,Z 669.497,A -85,B 0,C 180,E1 -9433.417,E2 -9433.417} C_VEL
LIN {X 0,Y 435.931,Z 682.757,A -85,B 0,C 180,E1 -9433.822,E2 -9433.822} C_VEL
LIN {X 0,Y 435.133,Z 696.091,A -85,B 0,C 180,E1 -9434.423,E2 -9434.423} C_VEL
LIN {X 0,Y 434.491,Z 707.347,A -85,B 0,C 180,E1 -9435.119,E2 -9435.119} C_VEL
LIN {X 0,Y 433.484,Z 724.112,A -85,B 0,C 180,E1 -9436.402,E2 -9436.402} C_VEL
LIN {X 0,Y 432.995,Z 735.064,A -85,B 0,C 180,E1 -9437.46,E2 -9437.46} C_VEL
LIN {X 0,Y 432.533,Z 742.186,A -85,B 0,C 180,E1 -9438.28,E2 -9438.28} C_VEL
LIN {X 0,Y 432.148,Z 750.712,A -85,B 0,C 180,E1 -9439.456,E2 -9439.456} C_VEL
LIN {X 0,Y 431.789,Z 759.053,A -85,B 0,C 180,E1 -9440.867,E2 -9440.867} C_VEL
LIN {X 0,Y 431.581,Z 764.705,A -85,B 0,C 180,E1 -9442.042,E2 -9442.042} C_VEL
LIN {X 0,Y 431.463,Z 770.483,A -85,B 0,C 180,E1 -9443.524,E2 -9443.524} C_VEL
LIN {X 0,Y 431.446,Z 774.507,A -85,B 0,C 180,E1 -9444.858,E2 -9444.858} C_VEL
LIN {X 0,Y 431.377,Z 777.662,A -85,B 0,C 180,E1 -9446.262,E2 -9446.262} C_VEL
LIN {X 0,Y 431.419,Z 779.178,A -85,B 0,C 180,E1 -9447.197,E2 -9447.197} C_VEL
LIN {X 0,Y 431.411,Z 780.254,A -85,B 0,C 180,E1 -9448.131,E2 -9448.131} C_VEL
LIN {X 0,Y 431.4,Z 780.918,A -85,B 0,C 180,E1 -9449.065,E2 -9449.065} C_VEL
LIN {X 0,Y 431.415,Z 781.145,A -85,B 0,C 180,E1 -9449.998,E2 -9449.998} C_VEL
LIN {X 0,Y 431.398,Z 780.913,A -85,B 0,C 180,E1 -9450.932,E2 -9450.932} C_VEL
LIN {X 0,Y 431.407,Z 780.273,A -85,B 0,C 180,E1 -9451.866,E2 -9451.866} C_VEL
LIN {X 0,Y 431.413,Z 779.215,A -85,B 0,C 180,E1 -9452.8,E2 -9452.8} C_VEL
LIN {X 0,Y 431.374,Z 777.669,A -85,B 0,C 180,E1 -9453.735,E2 -9453.735} C_VEL
LIN {X 0,Y 431.435,Z 774.513,A -85,B 0,C 180,E1 -9455.139,E2 -9455.139} C_VEL
LIN {X 0,Y 431.439,Z 770.222,A -85,B 0,C 180,E1 -9456.546,E2 -9456.546} C_VEL
LIN {X 0,Y 431.575,Z 764.683,A -85,B 0,C 180,E1 -9457.955,E2 -9457.955} C_VEL
LIN {X 0,Y 431.801,Z 757.713,A -85,B 0,C 180,E1 -9459.365,E2 -9459.365} C_VEL
LIN {X 0,Y 432.12,Z 750.562,A -85,B 0,C 180,E1 -9460.541,E2 -9460.541} C_VEL
LIN {X 0,Y 432.516,Z 741.865,A -85,B 0,C 180,E1 -9461.717,E2 -9461.717} C_VEL
LIN {X 0,Y 433.113,Z 732.311,A -85,B 0,C 180,E1 -9462.771,E2 -9462.771} C_VEL
LIN {X 0,Y 433.555,Z 720.709,A -85,B 0,C 180,E1 -9463.808,E2 -9463.808} C_VEL
LIN {X 0,Y 434.167,Z 708.511,A -85,B 0,C 180,E1 -9464.649,E2 -9464.649} C_VEL
LIN {X 0,Y 434.976,Z 693.473,A -85,B 0,C 180,E1 -9465.52,E2 -9465.52} C_VEL
LIN {X 0,Y 435.66,Z 680.259,A -85,B 0,C 180,E1 -9466.065,E2 -9466.065} C_VEL
LIN {X 0,Y 435.992,Z 667.001,A -85,B 0,C 180,E1 -9466.413,E2 -9466.413} C_VEL
LIN {X 0,Y 436.593,Z 590.559,A -85,B 0,C 180,E1 -9467.681,E2 -9467.681} C_VEL
LIN {X 0,Y 433.384,Z 559.83,A -85,B 0,C 180,E1 -9468.329,E2 -9468.329} C_VEL
LIN {X 0,Y 434.294,Z 536.575,A -85,B 0,C 180,E1 -9471.6,E2 -9471.6} C_VEL
LIN {X 0,Y 435.478,Z 514.136,A -85,B 0,C 180,E1 -9474.808,E2 -9474.808} C_VEL
LIN {X 0,Y 436.72,Z 491.545,A -85,B 0,C 180,E1 -9478.078,E2 -9478.078} C_VEL
LIN {X 0,Y 434.855,Z 481.798,A -85,B 0,C 180,E1 -9479.623,E2 -9479.623} C_VEL
LIN {X 0,Y 432.372,Z 470.736,A -85,B 0,C 180,E1 -9481.476,E2 -9481.476} C_VEL
LIN {X 0,Y 432.33,Z 470.633,A -85,B 0,C 180,E1 -9484.676,E2 -9484.676} C_VEL
LIN {X 0,Y 432.315,Z 470.637,A -85,B 0,C 180,E1 -9488.15,E2 -9488.15} C_VEL
LIN {X 0,Y 432.3,Z 470.634,A -85,B 0,C 180,E1 -9491.798,E2 -9491.798} C_VEL
LIN {X 0,Y 432.325,Z 470.634,A -85,B 0,C 180,E1 -9494.346,E2 -9494.346} C_VEL
LIN {X 0,Y 432.307,Z 470.631,A -85,B 0,C 180,E1 -9497.015,E2 -9497.015} C_VEL
LIN {X 0,Y 432.299,Z 470.634,A -85,B 0,C 180,E1 -9499.823,E2 -9499.823} C_VEL
LIN {X 0,Y 432.294,Z 470.632,A -85,B 0,C 180,E1 -9503.02,E2 -9503.02} C_VEL
LIN {X 0,Y 432.348,Z 470.629,A -85,B 0,C 180,E1 -9505.995,E2 -9505.995} C_VEL
LIN {X 0,Y 432.335,Z 470.627,A -85,B 0,C 180,E1 -9509.488,E2 -9509.488} C_VEL
LIN {X 0,Y 432.373,Z 470.624,A -85,B 0,C 180,E1 -9512.927,E2 -9512.927} C_VEL
LIN {X 0,Y 432.354,Z 470.628,A -85,B 0,C 180,E1 -9516.022,E2 -9516.022} C_VEL
LIN {X 0,Y 432.337,Z 470.628,A -85,B 0,C 180,E1 -9519.045,E2 -9519.045} C_VEL
LIN {X 0,Y 432.363,Z 470.626,A -85,B 0,C 180,E1 -9522.01,E2 -9522.01} C_VEL
LIN {X 0,Y 432.381,Z 470.623,A -85,B 0,C 180,E1 -9524.926,E2 -9524.926} C_VEL
LIN {X 0,Y 432.446,Z 470.614,A -85,B 0,C 180,E1 -9527.803,E2 -9527.803} C_VEL
LIN {X 0,Y 432.478,Z 470.609,A -85,B 0,C 180,E1 -9531.59,E2 -9531.59} C_VEL
LIN {X 0,Y 432.577,Z 470.603,A -85,B 0,C 180,E1 -9534.406,E2 -9534.406} C_VEL
LIN {X 0,Y 432.59,Z 470.598,A -85,B 0,C 180,E1 -9538.138,E2 -9538.138} C_VEL
LIN {X 0,Y 432.718,Z 470.581,A -85,B 0,C 180,E1 -9540,E2 -9540} C_VEL
LIN {X 0,Y 432.59,Z 470.6,A -85,B 0,C 180,E1 -9542.793,E2 -9542.793} C_VEL
LIN {X 0,Y 432.554,Z 470.607,A -85,B 0,C 180,E1 -9546.53,E2 -9546.53} C_VEL
LIN {X 0,Y 432.43,Z 470.616,A -85,B 0,C 180,E1 -9549.353,E2 -9549.353} C_VEL
LIN {X 0,Y 432.416,Z 470.622,A -85,B 0,C 180,E1 -9552.804,E2 -9552.804} C_VEL
LIN {X 0,Y 432.398,Z 470.624,A -85,B 0,C 180,E1 -9556.479,E2 -9556.479} C_VEL
LIN {X 0,Y 432.325,Z 470.629,A -85,B 0,C 180,E1 -9559.961,E2 -9559.961} C_VEL
LIN {X 0,Y 432.305,Z 470.635,A -85,B 0,C 180,E1 -9562.965,E2 -9562.965} C_VEL
LIN {X 0,Y 432.351,Z 470.626,A -85,B 0,C 180,E1 -9566.033,E2 -9566.033} C_VEL
LIN {X 0,Y 432.329,Z 470.63,A -85,B 0,C 180,E1 -9569.188,E2 -9569.188} C_VEL
LIN {X 0,Y 432.31,Z 470.633,A -85,B 0,C 180,E1 -9572.444,E2 -9572.444} C_VEL
LIN {X 0,Y 432.333,Z 470.627,A -85,B 0,C 180,E1 -9575.633,E2 -9575.633} C_VEL
LIN {X 0,Y 432.334,Z 470.633,A -85,B 0,C 180,E1 -9578.716,E2 -9578.716} C_VEL
LIN {X 0,Y 432.323,Z 470.628,A -85,B 0,C 180,E1 -9581.798,E2 -9581.798} C_VEL
LIN {X 0,Y 432.331,Z 470.629,A -85,B 0,C 180,E1 -9584.347,E2 -9584.347} C_VEL
LIN {X 0,Y 432.355,Z 470.631,A -85,B 0,C 180,E1 -9587.01,E2 -9587.01} C_VEL
LIN {X 0,Y 432.348,Z 470.625,A -85,B 0,C 180,E1 -9589.818,E2 -9589.818} C_VEL
LIN {X 0,Y 432.307,Z 470.637,A -85,B 0,C 180,E1 -9593.024,E2 -9593.024} C_VEL
LIN {X 0,Y 432.35,Z 470.625,A -85,B 0,C 180,E1 -9595.998,E2 -9595.998} C_VEL
LIN {X 0,Y 432.339,Z 470.628,A -85,B 0,C 180,E1 -9599.491,E2 -9599.491} C_VEL
LIN {X 0,Y 432.385,Z 470.628,A -85,B 0,C 180,E1 -9602.93,E2 -9602.93} C_VEL
LIN {X 0,Y 432.365,Z 470.623,A -85,B 0,C 180,E1 -9606.025,E2 -9606.025} C_VEL
LIN {X 0,Y 432.345,Z 470.634,A -85,B 0,C 180,E1 -9609.048,E2 -9609.048} C_VEL
LIN {X 0,Y 432.373,Z 470.622,A -85,B 0,C 180,E1 -9612.013,E2 -9612.013} C_VEL
LIN {X 0,Y 432.391,Z 470.625,A -85,B 0,C 180,E1 -9614.928,E2 -9614.928} C_VEL
LIN {X 0,Y 432.455,Z 470.613,A -85,B 0,C 180,E1 -9617.805,E2 -9617.805} C_VEL
LIN {X 0,Y 432.489,Z 470.613,A -85,B 0,C 180,E1 -9621.592,E2 -9621.592} C_VEL
LIN {X 0,Y 432.597,Z 470.6,A -85,B 0,C 180,E1 -9624.408,E2 -9624.408} C_VEL
LIN {X 0,Y 432.415,Z 470.752,A -85,B 0,C 180,E1 -9626.157,E2 -9626.157} C_VEL
LIN {X 0,Y 432.561,Z 471.576,A -85,B 0,C 180,E1 -9626.313,E2 -9626.313} C_VEL
LIN {X 0,Y 437.082,Z 483.913,A -85,B 0,C 180,E1 -9626.723,E2 -9626.723} C_VEL
LIN {X 0,Y 436.633,Z 528.362,A -85,B 0,C 180,E1 -9627.452,E2 -9627.452} C_VEL
LIN {X 0,Y 436.034,Z 534.21,A -85,B 0,C 180,E1 -9627.523,E2 -9627.523} C_VEL
LIN {X 0,Y 430.513,Z 553.206,A -85,B 0,C 180,E1 -9627.672,E2 -9627.672} C_VEL
LIN {X 0,Y 429.726,Z 558.966,A -85,B 0,C 180,E1 -9627.808,E2 -9627.808} C_VEL
LIN {X 0,Y 429.576,Z 571.771,A -85,B 0,C 180,E1 -9628.3,E2 -9628.3} C_VEL
LIN {X 0,Y 429.281,Z 583.699,A -85,B 0,C 180,E1 -9628.941,E2 -9628.941} C_VEL
LIN {X 0,Y 428.91,Z 594.52,A -85,B 0,C 180,E1 -9629.701,E2 -9629.701} C_VEL
LIN {X 0,Y 428.397,Z 605.529,A -85,B 0,C 180,E1 -9630.683,E2 -9630.683} C_VEL
LIN {X 0,Y 427.859,Z 614.357,A -85,B 0,C 180,E1 -9631.649,E2 -9631.649} C_VEL
LIN {X 0,Y 427.382,Z 623.195,A -85,B 0,C 180,E1 -9632.829,E2 -9632.829} C_VEL
LIN {X 0,Y 426.811,Z 631.862,A -85,B 0,C 180,E1 -9634.251,E2 -9634.251} C_VEL
LIN {X 0,Y 426.381,Z 638.783,A -85,B 0,C 180,E1 -9635.677,E2 -9635.677} C_VEL
LIN {X 0,Y 426.065,Z 644.316,A -85,B 0,C 180,E1 -9637.108,E2 -9637.108} C_VEL
LIN {X 0,Y 425.716,Z 648.697,A -85,B 0,C 180,E1 -9638.546,E2 -9638.546} C_VEL
LIN {X 0,Y 425.551,Z 651.016,A -85,B 0,C 180,E1 -9639.507,E2 -9639.507} C_VEL
LIN {X 0,Y 425.414,Z 652.91,A -85,B 0,C 180,E1 -9640.472,E2 -9640.472} C_VEL
LIN {X 0,Y 425.307,Z 654.336,A -85,B 0,C 180,E1 -9641.439,E2 -9641.439} C_VEL
LIN {X 0,Y 425.289,Z 655.692,A -85,B 0,C 180,E1 -9642.843,E2 -9642.843} C_VEL
LIN {X 0,Y 425.286,Z 656.196,A -85,B 0,C 180,E1 -9644.354,E2 -9644.354} C_VEL
LIN {X 0,Y 425.317,Z 655.979,A -85,B 0,C 180,E1 -9645.332,E2 -9645.332} C_VEL
LIN {X 0,Y 425.46,Z 655.072,A -85,B 0,C 180,E1 -9646.65,E2 -9646.65} C_VEL
LIN {X 0,Y 425.665,Z 652.858,A -85,B 0,C 180,E1 -9648.284,E2 -9648.284} C_VEL
LIN {X 0,Y 426.019,Z 649.46,A -85,B 0,C 180,E1 -9649.895,E2 -9649.895} C_VEL
LIN {X 0,Y 426.384,Z 645.551,A -85,B 0,C 180,E1 -9651.263,E2 -9651.263} C_VEL
LIN {X 0,Y 426.966,Z 639.247,A -85,B 0,C 180,E1 -9652.955,E2 -9652.955} C_VEL
LIN {X 0,Y 427.668,Z 631.656,A -85,B 0,C 180,E1 -9654.517,E2 -9654.517} C_VEL
LIN {X 0,Y 428.271,Z 623.963,A -85,B 0,C 180,E1 -9655.792,E2 -9655.792} C_VEL
LIN {X 0,Y 429.003,Z 614.699,A -85,B 0,C 180,E1 -9657.041,E2 -9657.041} C_VEL
LIN {X 0,Y 429.546,Z 605.756,A -85,B 0,C 180,E1 -9658.028,E2 -9658.028} C_VEL
LIN {X 0,Y 430.183,Z 595.462,A -85,B 0,C 180,E1 -9658.948,E2 -9658.948} C_VEL
LIN {X 0,Y 430.665,Z 584.134,A -85,B 0,C 180,E1 -9659.75,E2 -9659.75} C_VEL
LIN {X 0,Y 431.025,Z 571.409,A -85,B 0,C 180,E1 -9660.431,E2 -9660.431} C_VEL
LIN {X 0,Y 431.196,Z 559.128,A -85,B 0,C 180,E1 -9660.893,E2 -9660.893} C_VEL
LIN {X 0,Y 431.209,Z 544.682,A -85,B 0,C 180,E1 -9661.216,E2 -9661.216} C_VEL
LIN {X 0,Y 431.832,Z 487.626,A -85,B 0,C 180,E1 -9662.19,E2 -9662.19} C_VEL
LIN {X 0,Y 425.521,Z 472.56,A -85,B 0,C 180,E1 -9662.825,E2 -9662.825} C_VEL
LIN {X 0,Y 425.337,Z 471.613,A -85,B 0,C 180,E1 -9663.01,E2 -9663.01} C_VEL
LIN {X 0,Y 425.268,Z 471.512,A -85,B 0,C 180,E1 -9666.51,E2 -9666.51} C_VEL
LIN {X 0,Y 425.285,Z 471.506,A -85,B 0,C 180,E1 -9669.042,E2 -9669.042} C_VEL
LIN {X 0,Y 425.294,Z 471.505,A -85,B 0,C 180,E1 -9671.959,E2 -9671.959} C_VEL
LIN {X 0,Y 425.289,Z 471.511,A -85,B 0,C 180,E1 -9675.284,E2 -9675.284} C_VEL
LIN {X 0,Y 425.28,Z 471.512,A -85,B 0,C 180,E1 -9678.622,E2 -9678.622} C_VEL
LIN {X 0,Y 425.365,Z 471.695,A -85,B 0,C 180,E1 -9680.061,E2 -9680.061} C_VEL
LIN {X 0,Y 428.593,Z 487.061,A -85,B 0,C 180,E1 -9682.88,E2 -9682.88} C_VEL
LIN {X 0,Y 428.387,Z 497.668,A -85,B 0,C 180,E1 -9684.669,E2 -9684.669} C_VEL
LIN {X 0,Y 427.692,Z 515.826,A -85,B 0,C 180,E1 -9687.721,E2 -9687.721} C_VEL
LIN {X 0,Y 427.569,Z 520.738,A -85,B 0,C 180,E1 -9688.517,E2 -9688.517} C_VEL
LIN {X 0,Y 430.415,Z 537.517,A -85,B 0,C 180,E1 -9688.983,E2 -9688.983} C_VEL
LIN {X 0,Y 428.968,Z 631.082,A -85,B 0,C 180,E1 -9690.763,E2 -9690.763} C_VEL
LIN {X 0,Y 428.623,Z 644.306,A -85,B 0,C 180,E1 -9691.207,E2 -9691.207} C_VEL
LIN {X 0,Y 428.102,Z 657.144,A -85,B 0,C 180,E1 -9691.838,E2 -9691.838} C_VEL
LIN {X 0,Y 427.66,Z 668.823,A -85,B 0,C 180,E1 -9692.604,E2 -9692.604} C_VEL
LIN {X 0,Y 426.994,Z 680.763,A -85,B 0,C 180,E1 -9693.615,E2 -9693.615} C_VEL
LIN {X 0,Y 426.42,Z 690.374,A -85,B 0,C 180,E1 -9694.627,E2 -9694.627} C_VEL
LIN {X 0,Y 425.872,Z 700.144,A -85,B 0,C 180,E1 -9695.894,E2 -9695.894} C_VEL
LIN {X 0,Y 425.398,Z 708.058,A -85,B 0,C 180,E1 -9697.155,E2 -9697.155} C_VEL
LIN {X 0,Y 424.962,Z 715.723,A -85,B 0,C 180,E1 -9698.665,E2 -9698.665} C_VEL
LIN {X 0,Y 424.645,Z 721.884,A -85,B 0,C 180,E1 -9700.218,E2 -9700.218} C_VEL
LIN {X 0,Y 424.411,Z 726.322,A -85,B 0,C 180,E1 -9701.662,E2 -9701.662} C_VEL
LIN {X 0,Y 424.333,Z 728.727,A -85,B 0,C 180,E1 -9702.655,E2 -9702.655} C_VEL
LIN {X 0,Y 424.199,Z 731.074,A -85,B 0,C 180,E1 -9703.934,E2 -9703.934} C_VEL
LIN {X 0,Y 424.081,Z 733,A -85,B 0,C 180,E1 -9705.607,E2 -9705.607} C_VEL
LIN {X 0,Y 424.102,Z 733.503,A -85,B 0,C 180,E1 -9706.585,E2 -9706.585} C_VEL
LIN {X 0,Y 424.211,Z 733.535,A -85,B 0,C 180,E1 -9707.819,E2 -9707.819} C_VEL
LIN {X 0,Y 424.226,Z 732.433,A -85,B 0,C 180,E1 -9709.5,E2 -9709.5} C_VEL
LIN {X 0,Y 424.281,Z 731.203,A -85,B 0,C 180,E1 -9710.466,E2 -9710.466} C_VEL
LIN {X 0,Y 424.468,Z 728.538,A -85,B 0,C 180,E1 -9711.91,E2 -9711.91} C_VEL
LIN {X 0,Y 424.675,Z 724.828,A -85,B 0,C 180,E1 -9713.348,E2 -9713.348} C_VEL
LIN {X 0,Y 424.912,Z 719.982,A -85,B 0,C 180,E1 -9714.781,E2 -9714.781} C_VEL
LIN {X 0,Y 425.293,Z 713.847,A -85,B 0,C 180,E1 -9716.21,E2 -9716.21} C_VEL
LIN {X 0,Y 425.814,Z 706.141,A -85,B 0,C 180,E1 -9717.636,E2 -9717.636} C_VEL
LIN {X 0,Y 426.508,Z 696.595,A -85,B 0,C 180,E1 -9719.056,E2 -9719.056} C_VEL
LIN {X 0,Y 427.166,Z 686.633,A -85,B 0,C 180,E1 -9720.236,E2 -9720.236} C_VEL
LIN {X 0,Y 427.836,Z 675.539,A -85,B 0,C 180,E1 -9721.295,E2 -9721.295} C_VEL
LIN {X 0,Y 428.383,Z 664.693,A -85,B 0,C 180,E1 -9722.116,E2 -9722.116} C_VEL
LIN {X 0,Y 429.021,Z 651.456,A -85,B 0,C 180,E1 -9722.876,E2 -9722.876} C_VEL
LIN {X 0,Y 429.414,Z 638.725,A -85,B 0,C 180,E1 -9723.402,E2 -9723.402} C_VEL
LIN {X 0,Y 429.674,Z 625.48,A -85,B 0,C 180,E1 -9723.752,E2 -9723.752} C_VEL
LIN {X 0,Y 431.344,Z 538.062,A -85,B 0,C 180,E1 -9725.48,E2 -9725.48} C_VEL
LIN {X 0,Y 428.995,Z 525.318,A -85,B 0,C 180,E1 -9725.892,E2 -9725.892} C_VEL
LIN {X 0,Y 428.486,Z 522.667,A -85,B 0,C 180,E1 -9726.032,E2 -9726.032} C_VEL
LIN {X 0,Y 429.255,Z 499.419,A -85,B 0,C 180,E1 -9729.869,E2 -9729.869} C_VEL
LIN {X 0,Y 429.574,Z 490.455,A -85,B 0,C 180,E1 -9731.322,E2 -9731.322} C_VEL
LIN {X 0,Y 428.081,Z 482.104,A -85,B 0,C 180,E1 -9732.805,E2 -9732.805} C_VEL
LIN {X 0,Y 425.385,Z 471.64,A -85,B 0,C 180,E1 -9734.777,E2 -9734.777} C_VEL
LIN {X 0,Y 425.341,Z 471.506,A -85,B 0,C 180,E1 -9737.303,E2 -9737.303} C_VEL
LIN {X 0,Y 425.304,Z 471.508,A -85,B 0,C 180,E1 -9740.305,E2 -9740.305} C_VEL
LIN {X 0,Y 425.292,Z 471.509,A -85,B 0,C 180,E1 -9743.366,E2 -9743.366} C_VEL
LIN {X 0,Y 425.354,Z 471.502,A -85,B 0,C 180,E1 -9746.495,E2 -9746.495} C_VEL
LIN {X 0,Y 425.299,Z 471.506,A -85,B 0,C 180,E1 -9749.719,E2 -9749.719} C_VEL
LIN {X 0,Y 425.291,Z 471.51,A -85,B 0,C 180,E1 -9753.048,E2 -9753.048} C_VEL
LIN {X 0,Y 425.291,Z 471.507,A -85,B 0,C 180,E1 -9755.928,E2 -9755.928} C_VEL
LIN {X 0,Y 425.296,Z 471.509,A -85,B 0,C 180,E1 -9759.041,E2 -9759.041} C_VEL
LIN {X 0,Y 425.298,Z 471.508,A -85,B 0,C 180,E1 -9761.958,E2 -9761.958} C_VEL
LIN {X 0,Y 425.293,Z 471.508,A -85,B 0,C 180,E1 -9765.282,E2 -9765.282} C_VEL
LIN {X 0,Y 425.282,Z 471.51,A -85,B 0,C 180,E1 -9768.621,E2 -9768.621} C_VEL
LIN {X 0,Y 425.299,Z 471.491,A -85,B 0,C 180,E1 -9771.1,E2 -9771.1} C_VEL
LIN {X 0,Y 425.302,Z 471.503,A -85,B 0,C 180,E1 -9774.663,E2 -9774.663} C_VEL
LIN {X 0,Y 425.322,Z 471.697,A -85,B 0,C 180,E1 -9777.525,E2 -9777.525} C_VEL
LIN {X 0,Y 428.584,Z 484.797,A -85,B 0,C 180,E1 -9779.933,E2 -9779.933} C_VEL
LIN {X 0,Y 430.349,Z 493.714,A -85,B 0,C 180,E1 -9781.465,E2 -9781.465} C_VEL
LIN {X 0,Y 429.677,Z 505.475,A -85,B 0,C 180,E1 -9783.267,E2 -9783.267} C_VEL
LIN {X 0,Y 428.247,Z 527.332,A -85,B 0,C 180,E1 -9786.547,E2 -9786.547} C_VEL
LIN {X 0,Y 426.845,Z 552.569,A -85,B 0,C 180,E1 -9790.272,E2 -9790.272} C_VEL
LIN {X 0,Y 426.649,Z 557.78,A -85,B 0,C 180,E1 -9790.986,E2 -9790.986} C_VEL
LIN {X 0,Y 429.678,Z 583.816,A -85,B 0,C 180,E1 -9791.616,E2 -9791.616} C_VEL
LIN {X 0,Y 430.572,Z 594.629,A -85,B 0,C 180,E1 -9791.849,E2 -9791.849} C_VEL
LIN {X 0,Y 429.615,Z 668.583,A -85,B 0,C 180,E1 -9793.118,E2 -9793.118} C_VEL
LIN {X 0,Y 429.161,Z 681.807,A -85,B 0,C 180,E1 -9793.529,E2 -9793.529} C_VEL
LIN {X 0,Y 428.321,Z 694.555,A -85,B 0,C 180,E1 -9794.107,E2 -9794.107} C_VEL
LIN {X 0,Y 427.582,Z 706.756,A -85,B 0,C 180,E1 -9794.873,E2 -9794.873} C_VEL
LIN {X 0,Y 426.616,Z 722.851,A -85,B 0,C 180,E1 -9796.094,E2 -9796.094} C_VEL
LIN {X 0,Y 426.089,Z 733.695,A -85,B 0,C 180,E1 -9797.138,E2 -9797.138} C_VEL
LIN {X 0,Y 425.521,Z 741.846,A -85,B 0,C 180,E1 -9798.084,E2 -9798.084} C_VEL
LIN {X 0,Y 425.14,Z 750.371,A -85,B 0,C 180,E1 -9799.281,E2 -9799.281} C_VEL
LIN {X 0,Y 424.742,Z 758.715,A -85,B 0,C 180,E1 -9800.714,E2 -9800.714} C_VEL
LIN {X 0,Y 424.526,Z 764.362,A -85,B 0,C 180,E1 -9801.909,E2 -9801.909} C_VEL
LIN {X 0,Y 424.378,Z 770.528,A -85,B 0,C 180,E1 -9803.539,E2 -9803.539} C_VEL
LIN {X 0,Y 424.323,Z 775.285,A -85,B 0,C 180,E1 -9805.248,E2 -9805.248} C_VEL
LIN {X 0,Y 424.277,Z 777.287,A -85,B 0,C 180,E1 -9806.199,E2 -9806.199} C_VEL
LIN {X 0,Y 424.344,Z 778.795,A -85,B 0,C 180,E1 -9807.15,E2 -9807.15} C_VEL
LIN {X 0,Y 424.326,Z 779.867,A -85,B 0,C 180,E1 -9808.1,E2 -9808.1} C_VEL
LIN {X 0,Y 424.338,Z 780.528,A -85,B 0,C 180,E1 -9809.049,E2 -9809.049} C_VEL
LIN {X 0,Y 424.349,Z 780.743,A -85,B 0,C 180,E1 -9809.998,E2 -9809.998} C_VEL
LIN {X 0,Y 424.335,Z 780.507,A -85,B 0,C 180,E1 -9810.947,E2 -9810.947} C_VEL
LIN {X 0,Y 424.322,Z 779.858,A -85,B 0,C 180,E1 -9811.897,E2 -9811.897} C_VEL
LIN {X 0,Y 424.339,Z 778.787,A -85,B 0,C 180,E1 -9812.846,E2 -9812.846} C_VEL
LIN {X 0,Y 424.273,Z 776.304,A -85,B 0,C 180,E1 -9814.273,E2 -9814.273} C_VEL
LIN {X 0,Y 424.322,Z 772.757,A -85,B 0,C 180,E1 -9815.702,E2 -9815.702} C_VEL
LIN {X 0,Y 424.415,Z 768.03,A -85,B 0,C 180,E1 -9817.133,E2 -9817.133} C_VEL
LIN {X 0,Y 424.587,Z 761.982,A -85,B 0,C 180,E1 -9818.566,E2 -9818.566} C_VEL
LIN {X 0,Y 424.874,Z 754.403,A -85,B 0,C 180,E1 -9820,E2 -9820} C_VEL
LIN {X 0,Y 425.273,Z 746.635,A -85,B 0,C 180,E1 -9821.195,E2 -9821.195} C_VEL
LIN {X 0,Y 425.732,Z 737.12,A -85,B 0,C 180,E1 -9822.391,E2 -9822.391} C_VEL
LIN {X 0,Y 426.202,Z 727.585,A -85,B 0,C 180,E1 -9823.368,E2 -9823.368} C_VEL
LIN {X 0,Y 426.781,Z 716.316,A -85,B 0,C 180,E1 -9824.299,E2 -9824.299} C_VEL
LIN {X 0,Y 427.62,Z 701.424,A -85,B 0,C 180,E1 -9825.244,E2 -9825.244} C_VEL
LIN {X 0,Y 428.244,Z 689.361,A -85,B 0,C 180,E1 -9825.892,E2 -9825.892} C_VEL
LIN {X 0,Y 428.897,Z 675.47,A -85,B 0,C 180,E1 -9826.417,E2 -9826.417} C_VEL
LIN {X 0,Y 429.169,Z 662.663,A -85,B 0,C 180,E1 -9826.713,E2 -9826.713} C_VEL
LIN {X 0,Y 429.76,Z 591.334,A -85,B 0,C 180,E1 -9827.907,E2 -9827.907} C_VEL
LIN {X 0,Y 426.378,Z 559.114,A -85,B 0,C 180,E1 -9828.591,E2 -9828.591} C_VEL
LIN {X 0,Y 426.442,Z 555.945,A -85,B 0,C 180,E1 -9828.993,E2 -9828.993} C_VEL
LIN {X 0,Y 427.501,Z 533.642,A -85,B 0,C 180,E1 -9832.215,E2 -9832.215} C_VEL
LIN {X 0,Y 428.892,Z 508.463,A -85,B 0,C 180,E1 -9835.886,E2 -9835.886} C_VEL
LIN {X 0,Y 429.732,Z 492.071,A -85,B 0,C 180,E1 -9838.31,E2 -9838.31} C_VEL
LIN {X 0,Y 426.272,Z 475.763,A -85,B 0,C 180,E1 -9840.981,E2 -9840.981} C_VEL
LIN {X 0,Y 425.332,Z 471.613,A -85,B 0,C 180,E1 -9841.725,E2 -9841.725} C_VEL
LIN {X 0,Y 425.29,Z 471.509,A -85,B 0,C 180,E1 -9845.334,E2 -9845.334} C_VEL
LIN {X 0,Y 425.269,Z 471.508,A -85,B 0,C 180,E1 -9848.899,E2 -9848.899} C_VEL
LIN {X 0,Y 425.252,Z 471.512,A -85,B 0,C 180,E1 -9852.653,E2 -9852.653} C_VEL
LIN {X 0,Y 425.276,Z 471.506,A -85,B 0,C 180,E1 -9855.282,E2 -9855.282} C_VEL
LIN {X 0,Y 425.248,Z 471.513,A -85,B 0,C 180,E1 -9858.618,E2 -9858.618} C_VEL
LIN {X 0,Y 425.27,Z 471.507,A -85,B 0,C 180,E1 -9861.098,E2 -9861.098} C_VEL
LIN {X 0,Y 425.288,Z 471.508,A -85,B 0,C 180,E1 -9864.663,E2 -9864.663} C_VEL
LIN {X 0,Y 425.254,Z 471.514,A -85,B 0,C 180,E1 -9868.072,E2 -9868.072} C_VEL
LIN {X 0,Y 425.319,Z 471.501,A -85,B 0,C 180,E1 -9871.367,E2 -9871.367} C_VEL
LIN {X 0,Y 425.272,Z 471.512,A -85,B 0,C 180,E1 -9874.553,E2 -9874.553} C_VEL
LIN {X 0,Y 425.291,Z 471.509,A -85,B 0,C 180,E1 -9876.634,E2 -9876.634} C_VEL
LIN {X 0,Y 425.315,Z 471.509,A -85,B 0,C 180,E1 -9880.363,E2 -9880.363} C_VEL
LIN {X 0,Y 425.375,Z 471.494,A -85,B 0,C 180,E1 -9883.687,E2 -9883.687} C_VEL
LIN {X 0,Y 425.399,Z 471.491,A -85,B 0,C 180,E1 -9887.597,E2 -9887.597} C_VEL
LIN {X 0,Y 425.429,Z 471.487,A -85,B 0,C 180,E1 -9891.449,E2 -9891.449} C_VEL
LIN {X 0,Y 425.534,Z 471.479,A -85,B 0,C 180,E1 -9894.313,E2 -9894.313} C_VEL
LIN {X 0,Y 425.56,Z 471.473,A -85,B 0,C 180,E1 -9898.107,E2 -9898.107} C_VEL
LIN {X 0,Y 425.688,Z 471.457,A -85,B 0,C 180,E1 -9900,E2 -9900} C_VEL
LIN {X 0,Y 425.542,Z 471.477,A -85,B 0,C 180,E1 -9902.84,E2 -9902.84} C_VEL
LIN {X 0,Y 425.513,Z 471.484,A -85,B 0,C 180,E1 -9906.639,E2 -9906.639} C_VEL
LIN {X 0,Y 425.388,Z 471.492,A -85,B 0,C 180,E1 -9909.509,E2 -9909.509} C_VEL
LIN {X 0,Y 425.379,Z 471.498,A -85,B 0,C 180,E1 -9912.904,E2 -9912.904} C_VEL
LIN {X 0,Y 425.347,Z 471.504,A -85,B 0,C 180,E1 -9916.605,E2 -9916.605} C_VEL
LIN {X 0,Y 425.314,Z 471.501,A -85,B 0,C 180,E1 -9919.636,E2 -9919.636} C_VEL
LIN {X 0,Y 425.293,Z 471.505,A -85,B 0,C 180,E1 -9923.366,E2 -9923.366} C_VEL
LIN {X 0,Y 425.337,Z 471.505,A -85,B 0,C 180,E1 -9926.846,E2 -9926.846} C_VEL
LIN {X 0,Y 425.277,Z 471.506,A -85,B 0,C 180,E1 -9929.72,E2 -9929.72} C_VEL
LIN {X 0,Y 425.269,Z 471.512,A -85,B 0,C 180,E1 -9933.049,E2 -9933.049} C_VEL
LIN {X 0,Y 425.272,Z 471.507,A -85,B 0,C 180,E1 -9935.93,E2 -9935.93} C_VEL
LIN {X 0,Y 425.284,Z 471.51,A -85,B 0,C 180,E1 -9939.044,E2 -9939.044} C_VEL
LIN {X 0,Y 425.267,Z 471.512,A -85,B 0,C 180,E1 -9942.654,E2 -9942.654} C_VEL
LIN {X 0,Y 425.308,Z 471.502,A -85,B 0,C 180,E1 -9946.053,E2 -9946.053} C_VEL
LIN {X 0,Y 425.3,Z 471.507,A -85,B 0,C 180,E1 -9948.627,E2 -9948.627} C_VEL
LIN {X 0,Y 425.314,Z 471.507,A -85,B 0,C 180,E1 -9951.106,E2 -9951.106} C_VEL
LIN {X 0,Y 425.291,Z 471.508,A -85,B 0,C 180,E1 -9954.666,E2 -9954.666} C_VEL
LIN {X 0,Y 425.256,Z 471.509,A -85,B 0,C 180,E1 -9958.075,E2 -9958.075} C_VEL
LIN {X 0,Y 425.323,Z 471.504,A -85,B 0,C 180,E1 -9961.369,E2 -9961.369} C_VEL
LIN {X 0,Y 425.288,Z 471.507,A -85,B 0,C 180,E1 -9964.556,E2 -9964.556} C_VEL
LIN {X 0,Y 425.281,Z 471.507,A -85,B 0,C 180,E1 -9967.663,E2 -9967.663} C_VEL
LIN {X 0,Y 425.356,Z 471.499,A -85,B 0,C 180,E1 -9970.706,E2 -9970.706} C_VEL
LIN {X 0,Y 425.383,Z 471.494,A -85,B 0,C 180,E1 -9973.69,E2 -9973.69} C_VEL
LIN {X 0,Y 425.408,Z 471.492,A -85,B 0,C 180,E1 -9977.6,E2 -9977.6} C_VEL
LIN {X 0,Y 425.439,Z 471.492,A -85,B 0,C 180,E1 -9981.452,E2 -9981.452} C_VEL
LIN {X 0,Y 425.553,Z 471.478,A -85,B 0,C 180,E1 -9984.315,E2 -9984.315} C_VEL
LIN {X 0,Y 425.387,Z 471.658,A -85,B 0,C 180,E1 -9985.916,E2 -9985.916} C_VEL
LIN {X 0,Y 425.545,Z 472.527,A -85,B 0,C 180,E1 -9986.066,E2 -9986.066} C_VEL
LIN {X 0,Y 430.194,Z 485.146,A -85,B 0,C 180,E1 -9986.484,E2 -9986.484} C_VEL
LIN {X 0,Y 429.717,Z 553.31,A -85,B 0,C 180,E1 -9987.651,E2 -9987.651} C_VEL
LIN {X 0,Y 429.726,Z 558.966,A -85,B 0,C 180,E1 -9987.808,E2 -9987.808} C_VEL
LIN {X 0,Y 428.43,Z 566.578,A -85,B 0,C 180,E1 -9988.031,E2 -9988.031} C_VEL
LIN {X 0,Y 425.969,Z 573.949,A -85,B 0,C 180,E1 -9988.265,E2 -9988.265} C_VEL
LIN {X 0,Y 423.058,Z 582.963,A -85,B 0,C 180,E1 -9988.651,E2 -9988.651} C_VEL
LIN {X 0,Y 422.31,Z 588.278,A -85,B 0,C 180,E1 -9988.973,E2 -9988.973} C_VEL
LIN {X 0,Y 421.831,Z 599.677,A -85,B 0,C 180,E1 -9989.859,E2 -9989.859} C_VEL
LIN {X 0,Y 421.31,Z 609.721,A -85,B 0,C 180,E1 -9990.838,E2 -9990.838} C_VEL
LIN {X 0,Y 420.815,Z 618.713,A -85,B 0,C 180,E1 -9991.916,E2 -9991.916} C_VEL
LIN {X 0,Y 420.153,Z 628.436,A -85,B 0,C 180,E1 -9993.358,E2 -9993.358} C_VEL
LIN {X 0,Y 419.647,Z 636.253,A -85,B 0,C 180,E1 -9994.805,E2 -9994.805} C_VEL
LIN {X 0,Y 419.225,Z 642.501,A -85,B 0,C 180,E1 -9996.257,E2 -9996.257} C_VEL
LIN {X 0,Y 418.89,Z 647.478,A -85,B 0,C 180,E1 -9997.715,E2 -9997.715} C_VEL
LIN {X 0,Y 418.595,Z 651.349,A -85,B 0,C 180,E1 -9999.179,E2 -9999.179} C_VEL
LIN {X 0,Y 418.361,Z 654.2,A -85,B 0,C 180,E1 -10000.65,E2 -10000.65} C_VEL
LIN {X 0,Y 418.273,Z 656.496,A -85,B 0,C 180,E1 -10002.618,E2 -10002.618} C_VEL
LIN {X 0,Y 418.243,Z 657.049,A -85,B 0,C 180,E1 -10003.608,E2 -10003.608} C_VEL
LIN {X 0,Y 418.274,Z 657.158,A -85,B 0,C 180,E1 -10004.6,E2 -10004.6} C_VEL
LIN {X 0,Y 418.313,Z 656.88,A -85,B 0,C 180,E1 -10005.595,E2 -10005.595} C_VEL
LIN {X 0,Y 418.453,Z 655.994,A -85,B 0,C 180,E1 -10006.8,E2 -10006.8} C_VEL
LIN {X 0,Y 418.709,Z 653.497,A -85,B 0,C 180,E1 -10008.599,E2 -10008.599} C_VEL
LIN {X 0,Y 419.071,Z 650.313,A -85,B 0,C 180,E1 -10010.093,E2 -10010.093} C_VEL
LIN {X 0,Y 419.539,Z 645.893,A -85,B 0,C 180,E1 -10011.627,E2 -10011.627} C_VEL
LIN {X 0,Y 420.14,Z 639.712,A -85,B 0,C 180,E1 -10013.27,E2 -10013.27} C_VEL
LIN {X 0,Y 420.811,Z 632.932,A -85,B 0,C 180,E1 -10014.68,E2 -10014.68} C_VEL
LIN {X 0,Y 421.428,Z 625.557,A -85,B 0,C 180,E1 -10015.936,E2 -10015.936} C_VEL
LIN {X 0,Y 422.193,Z 616.104,A -85,B 0,C 180,E1 -10017.245,E2 -10017.245} C_VEL
LIN {X 0,Y 422.798,Z 607.33,A -85,B 0,C 180,E1 -10018.238,E2 -10018.238} C_VEL
LIN {X 0,Y 423.47,Z 597.131,A -85,B 0,C 180,E1 -10019.179,E2 -10019.179} C_VEL
LIN {X 0,Y 423.964,Z 585.901,A -85,B 0,C 180,E1 -10020.002,E2 -10020.002} C_VEL
LIN {X 0,Y 424.341,Z 573.595,A -85,B 0,C 180,E1 -10020.686,E2 -10020.686} C_VEL
LIN {X 0,Y 424.532,Z 561.226,A -85,B 0,C 180,E1 -10021.178,E2 -10021.178} C_VEL
LIN {X 0,Y 424.545,Z 547.464,A -85,B 0,C 180,E1 -10021.51,E2 -10021.51} C_VEL
LIN {X 0,Y 425.132,Z 488.896,A -85,B 0,C 180,E1 -10022.532,E2 -10022.532} C_VEL
LIN {X 0,Y 418.434,Z 473.243,A -85,B 0,C 180,E1 -10023.228,E2 -10023.228} C_VEL
LIN {X 0,Y 418.266,Z 472.437,A -85,B 0,C 180,E1 -10023.451,E2 -10023.451} C_VEL
LIN {X 0,Y 418.248,Z 472.389,A -85,B 0,C 180,E1 -10026.239,E2 -10026.239} C_VEL
LIN {X 0,Y 418.248,Z 472.38,A -85,B 0,C 180,E1 -10029.684,E2 -10029.684} C_VEL
LIN {X 0,Y 418.233,Z 472.382,A -85,B 0,C 180,E1 -10032.322,E2 -10032.322} C_VEL
LIN {X 0,Y 418.24,Z 472.389,A -85,B 0,C 180,E1 -10035.11,E2 -10035.11} C_VEL
LIN {X 0,Y 418.245,Z 472.388,A -85,B 0,C 180,E1 -10037.768,E2 -10037.768} C_VEL
LIN {X 0,Y 418.314,Z 472.608,A -85,B 0,C 180,E1 -10039.816,E2 -10039.816} C_VEL
LIN {X 0,Y 421.193,Z 486.16,A -85,B 0,C 180,E1 -10042.33,E2 -10042.33} C_VEL
LIN {X 0,Y 421.788,Z 490.71,A -85,B 0,C 180,E1 -10043.142,E2 -10043.142} C_VEL
LIN {X 0,Y 421.019,Z 511.019,A -85,B 0,C 180,E1 -10046.581,E2 -10046.581} C_VEL
LIN {X 0,Y 420.657,Z 521.103,A -85,B 0,C 180,E1 -10048.247,E2 -10048.247} C_VEL
LIN {X 0,Y 423.58,Z 538.924,A -85,B 0,C 180,E1 -10048.748,E2 -10048.748} C_VEL
LIN {X 0,Y 422.083,Z 631.446,A -85,B 0,C 180,E1 -10050.547,E2 -10050.547} C_VEL
LIN {X 0,Y 421.748,Z 643.91,A -85,B 0,C 180,E1 -10050.966,E2 -10050.966} C_VEL
LIN {X 0,Y 421.196,Z 656.907,A -85,B 0,C 180,E1 -10051.606,E2 -10051.606} C_VEL
LIN {X 0,Y 420.702,Z 669.312,A -85,B 0,C 180,E1 -10052.428,E2 -10052.428} C_VEL
LIN {X 0,Y 420.045,Z 680.784,A -85,B 0,C 180,E1 -10053.413,E2 -10053.413} C_VEL
LIN {X 0,Y 419.366,Z 691.903,A -85,B 0,C 180,E1 -10054.61,E2 -10054.61} C_VEL
LIN {X 0,Y 418.742,Z 702.018,A -85,B 0,C 180,E1 -10055.984,E2 -10055.984} C_VEL
LIN {X 0,Y 418.306,Z 709.698,A -85,B 0,C 180,E1 -10057.268,E2 -10057.268} C_VEL
LIN {X 0,Y 417.842,Z 717.077,A -85,B 0,C 180,E1 -10058.8,E2 -10058.8} C_VEL
LIN {X 0,Y 417.511,Z 723.462,A -85,B 0,C 180,E1 -10060.505,E2 -10060.505} C_VEL
LIN {X 0,Y 417.321,Z 727.312,A -85,B 0,C 180,E1 -10061.848,E2 -10061.848} C_VEL
LIN {X 0,Y 417.16,Z 730.553,A -85,B 0,C 180,E1 -10063.358,E2 -10063.358} C_VEL
LIN {X 0,Y 417.07,Z 732.095,A -85,B 0,C 180,E1 -10064.359,E2 -10064.359} C_VEL
LIN {X 0,Y 416.997,Z 733.172,A -85,B 0,C 180,E1 -10065.357,E2 -10065.357} C_VEL
LIN {X 0,Y 417.009,Z 733.826,A -85,B 0,C 180,E1 -10066.353,E2 -10066.353} C_VEL
LIN {X 0,Y 417.115,Z 733.958,A -85,B 0,C 180,E1 -10067.759,E2 -10067.759} C_VEL
LIN {X 0,Y 417.131,Z 733.097,A -85,B 0,C 180,E1 -10069.32,E2 -10069.32} C_VEL
LIN {X 0,Y 417.184,Z 731.982,A -85,B 0,C 180,E1 -10070.302,E2 -10070.302} C_VEL
LIN {X 0,Y 417.293,Z 730.42,A -85,B 0,C 180,E1 -10071.282,E2 -10071.282} C_VEL
LIN {X 0,Y 417.523,Z 727.116,A -85,B 0,C 180,E1 -10072.796,E2 -10072.796} C_VEL
LIN {X 0,Y 417.728,Z 722.988,A -85,B 0,C 180,E1 -10074.207,E2 -10074.207} C_VEL
LIN {X 0,Y 418.11,Z 717.525,A -85,B 0,C 180,E1 -10075.662,E2 -10075.662} C_VEL
LIN {X 0,Y 418.546,Z 710.674,A -85,B 0,C 180,E1 -10077.113,E2 -10077.113} C_VEL
LIN {X 0,Y 419.229,Z 702.093,A -85,B 0,C 180,E1 -10078.559,E2 -10078.559} C_VEL
LIN {X 0,Y 419.867,Z 693.327,A -85,B 0,C 180,E1 -10079.761,E2 -10079.761} C_VEL
LIN {X 0,Y 420.557,Z 683.66,A -85,B 0,C 180,E1 -10080.838,E2 -10080.838} C_VEL
LIN {X 0,Y 421.216,Z 673.074,A -85,B 0,C 180,E1 -10081.793,E2 -10081.793} C_VEL
LIN {X 0,Y 421.822,Z 661.454,A -85,B 0,C 180,E1 -10082.626,E2 -10082.626} C_VEL
LIN {X 0,Y 422.343,Z 649.944,A -85,B 0,C 180,E1 -10083.256,E2 -10083.256} C_VEL
LIN {X 0,Y 422.761,Z 636.402,A -85,B 0,C 180,E1 -10083.786,E2 -10083.786} C_VEL
LIN {X 0,Y 423.085,Z 621.139,A -85,B 0,C 180,E1 -10084.148,E2 -10084.148} C_VEL
LIN {X 0,Y 424.734,Z 538.289,A -85,B 0,C 180,E1 -10085.846,E2 -10085.846} C_VEL
LIN {X 0,Y 421.906,Z 524.157,A -85,B 0,C 180,E1 -10086.337,E2 -10086.337} C_VEL
LIN {X 0,Y 421.742,Z 522.844,A -85,B 0,C 180,E1 -10086.459,E2 -10086.459} C_VEL
LIN {X 0,Y 422.478,Z 502.712,A -85,B 0,C 180,E1 -10089.818,E2 -10089.818} C_VEL
LIN {X 0,Y 422.909,Z 492.488,A -85,B 0,C 180,E1 -10091.503,E2 -10091.503} C_VEL
LIN {X 0,Y 421.351,Z 484.091,A -85,B 0,C 180,E1 -10093.014,E2 -10093.014} C_VEL
LIN {X 0,Y 418.329,Z 472.499,A -85,B 0,C 180,E1 -10095.25,E2 -10095.25} C_VEL
LIN {X 0,Y 418.287,Z 472.383,A -85,B 0,C 180,E1 -10097.604,E2 -10097.604} C_VEL
LIN {X 0,Y 418.258,Z 472.387,A -85,B 0,C 180,E1 -10100.663,E2 -10100.663} C_VEL
LIN {X 0,Y 418.282,Z 472.382,A -85,B 0,C 180,E1 -10103.782,E2 -10103.782} C_VEL
LIN {X 0,Y 418.319,Z 472.379,A -85,B 0,C 180,E1 -10107.07,E2 -10107.07} C_VEL
LIN {X 0,Y 418.253,Z 472.384,A -85,B 0,C 180,E1 -10110.272,E2 -10110.272} C_VEL
LIN {X 0,Y 418.257,Z 472.383,A -85,B 0,C 180,E1 -10113.677,E2 -10113.677} C_VEL
LIN {X 0,Y 418.248,Z 472.386,A -85,B 0,C 180,E1 -10117.224,E2 -10117.224} C_VEL
LIN {X 0,Y 418.255,Z 472.384,A -85,B 0,C 180,E1 -10119.682,E2 -10119.682} C_VEL
LIN {X 0,Y 418.238,Z 472.387,A -85,B 0,C 180,E1 -10122.321,E2 -10122.321} C_VEL
LIN {X 0,Y 418.244,Z 472.387,A -85,B 0,C 180,E1 -10125.108,E2 -10125.108} C_VEL
LIN {X 0,Y 418.248,Z 472.387,A -85,B 0,C 180,E1 -10127.766,E2 -10127.766} C_VEL
LIN {X 0,Y 418.25,Z 472.374,A -85,B 0,C 180,E1 -10130.62,E2 -10130.62} C_VEL
LIN {X 0,Y 418.249,Z 472.389,A -85,B 0,C 180,E1 -10133.975,E2 -10133.975} C_VEL
LIN {X 0,Y 418.261,Z 472.552,A -85,B 0,C 180,E1 -10137.135,E2 -10137.135} C_VEL
LIN {X 0,Y 421.732,Z 486.316,A -85,B 0,C 180,E1 -10139.727,E2 -10139.727} C_VEL
LIN {X 0,Y 423.456,Z 494.83,A -85,B 0,C 180,E1 -10141.228,E2 -10141.228} C_VEL
LIN {X 0,Y 423.286,Z 500.321,A -85,B 0,C 180,E1 -10142.1,E2 -10142.1} C_VEL
LIN {X 0,Y 421.737,Z 521.639,A -85,B 0,C 180,E1 -10145.378,E2 -10145.378} C_VEL
LIN {X 0,Y 420.284,Z 545.118,A -85,B 0,C 180,E1 -10148.928,E2 -10148.928} C_VEL
LIN {X 0,Y 419.695,Z 556.595,A -85,B 0,C 180,E1 -10150.608,E2 -10150.608} C_VEL
LIN {X 0,Y 422.259,Z 577.198,A -85,B 0,C 180,E1 -10151.139,E2 -10151.139} C_VEL
LIN {X 0,Y 423.886,Z 594.806,A -85,B 0,C 180,E1 -10151.533,E2 -10151.533} C_VEL
LIN {X 0,Y 422.881,Z 667.893,A -85,B 0,C 180,E1 -10152.81,E2 -10152.81} C_VEL
LIN {X 0,Y 422.368,Z 681.744,A -85,B 0,C 180,E1 -10153.256,E2 -10153.256} C_VEL
LIN {X 0,Y 421.497,Z 694.218,A -85,B 0,C 180,E1 -10153.843,E2 -10153.843} C_VEL
LIN {X 0,Y 420.713,Z 706.225,A -85,B 0,C 180,E1 -10154.62,E2 -10154.62} C_VEL
LIN {X 0,Y 419.907,Z 719.553,A -85,B 0,C 180,E1 -10155.595,E2 -10155.595} C_VEL
LIN {X 0,Y 419.31,Z 730.726,A -85,B 0,C 180,E1 -10156.629,E2 -10156.629} C_VEL
LIN {X 0,Y 418.608,Z 739.67,A -85,B 0,C 180,E1 -10157.638,E2 -10157.638} C_VEL
LIN {X 0,Y 418.199,Z 748.519,A -85,B 0,C 180,E1 -10158.855,E2 -10158.855} C_VEL
LIN {X 0,Y 417.75,Z 757.091,A -85,B 0,C 180,E1 -10160.313,E2 -10160.313} C_VEL
LIN {X 0,Y 417.454,Z 764.019,A -85,B 0,C 180,E1 -10161.771,E2 -10161.771} C_VEL
LIN {X 0,Y 417.271,Z 769.529,A -85,B 0,C 180,E1 -10163.228,E2 -10163.228} C_VEL
LIN {X 0,Y 417.255,Z 773.787,A -85,B 0,C 180,E1 -10164.683,E2 -10164.683} C_VEL
LIN {X 0,Y 417.179,Z 776.921,A -85,B 0,C 180,E1 -10166.135,E2 -10166.135} C_VEL
LIN {X 0,Y 417.27,Z 778.419,A -85,B 0,C 180,E1 -10167.102,E2 -10167.102} C_VEL
LIN {X 0,Y 417.244,Z 779.484,A -85,B 0,C 180,E1 -10168.068,E2 -10168.068} C_VEL
LIN {X 0,Y 417.247,Z 780.141,A -85,B 0,C 180,E1 -10169.033,E2 -10169.033} C_VEL
LIN {X 0,Y 417.285,Z 780.335,A -85,B 0,C 180,E1 -10169.998,E2 -10169.998} C_VEL
LIN {X 0,Y 417.274,Z 780.088,A -85,B 0,C 180,E1 -10170.963,E2 -10170.963} C_VEL
LIN {X 0,Y 417.241,Z 779.427,A -85,B 0,C 180,E1 -10171.929,E2 -10171.929} C_VEL
LIN {X 0,Y 417.266,Z 778.334,A -85,B 0,C 180,E1 -10172.895,E2 -10172.895} C_VEL
LIN {X 0,Y 417.191,Z 775.822,A -85,B 0,C 180,E1 -10174.346,E2 -10174.346} C_VEL
LIN {X 0,Y 417.222,Z 772.234,A -85,B 0,C 180,E1 -10175.799,E2 -10175.799} C_VEL
LIN {X 0,Y 417.344,Z 767.463,A -85,B 0,C 180,E1 -10177.254,E2 -10177.254} C_VEL
LIN {X 0,Y 417.525,Z 761.362,A -85,B 0,C 180,E1 -10178.712,E2 -10178.712} C_VEL
LIN {X 0,Y 417.822,Z 753.719,A -85,B 0,C 180,E1 -10180.171,E2 -10180.171} C_VEL
LIN {X 0,Y 418.229,Z 745.876,A -85,B 0,C 180,E1 -10181.386,E2 -10181.386} C_VEL
LIN {X 0,Y 418.681,Z 737.329,A -85,B 0,C 180,E1 -10182.48,E2 -10182.48} C_VEL
LIN {X 0,Y 419.172,Z 727.849,A -85,B 0,C 180,E1 -10183.479,E2 -10183.479} C_VEL
LIN {X 0,Y 419.761,Z 716.793,A -85,B 0,C 180,E1 -10184.42,E2 -10184.42} C_VEL
LIN {X 0,Y 420.397,Z 705.055,A -85,B 0,C 180,E1 -10185.202,E2 -10185.202} C_VEL
LIN {X 0,Y 421.311,Z 688.943,A -85,B 0,C 180,E1 -10186.099,E2 -10186.099} C_VEL
LIN {X 0,Y 421.98,Z 675.28,A -85,B 0,C 180,E1 -10186.632,E2 -10186.632} C_VEL
LIN {X 0,Y 422.289,Z 661.428,A -85,B 0,C 180,E1 -10186.962,E2 -10186.962} C_VEL
LIN {X 0,Y 422.892,Z 591.851,A -85,B 0,C 180,E1 -10188.146,E2 -10188.146} C_VEL
LIN {X 0,Y 419.395,Z 557.959,A -85,B 0,C 180,E1 -10188.881,E2 -10188.881} C_VEL
LIN {X 0,Y 420.511,Z 534.13,A -85,B 0,C 180,E1 -10192.345,E2 -10192.345} C_VEL
LIN {X 0,Y 421.938,Z 509.483,A -85,B 0,C 180,E1 -10196.003,E2 -10196.003} C_VEL
LIN {X 0,Y 422.845,Z 494.494,A -85,B 0,C 180,E1 -10198.248,E2 -10198.248} C_VEL
LIN {X 0,Y 421.591,Z 487.435,A -85,B 0,C 180,E1 -10199.401,E2 -10199.401} C_VEL
LIN {X 0,Y 418.285,Z 472.506,A -85,B 0,C 180,E1 -10201.971,E2 -10201.971} C_VEL
LIN {X 0,Y 418.251,Z 472.387,A -85,B 0,C 180,E1 -10204.839,E2 -10204.839} C_VEL
LIN {X 0,Y 418.227,Z 472.389,A -85,B 0,C 180,E1 -10208.442,E2 -10208.442} C_VEL
LIN {X 0,Y 418.215,Z 472.393,A -85,B 0,C 180,E1 -10212.234,E2 -10212.234} C_VEL
LIN {X 0,Y 418.227,Z 472.384,A -85,B 0,C 180,E1 -10215.107,E2 -10215.107} C_VEL
LIN {X 0,Y 418.223,Z 472.387,A -85,B 0,C 180,E1 -10217.764,E2 -10217.764} C_VEL
LIN {X 0,Y 418.227,Z 472.385,A -85,B 0,C 180,E1 -10221.555,E2 -10221.555} C_VEL
LIN {X 0,Y 418.248,Z 472.382,A -85,B 0,C 180,E1 -10225.158,E2 -10225.158} C_VEL
LIN {X 0,Y 418.234,Z 472.384,A -85,B 0,C 180,E1 -10227.471,E2 -10227.471} C_VEL
LIN {X 0,Y 418.257,Z 472.382,A -85,B 0,C 180,E1 -10230.894,E2 -10230.894} C_VEL
LIN {X 0,Y 418.249,Z 472.386,A -85,B 0,C 180,E1 -10234.094,E2 -10234.094} C_VEL
LIN {X 0,Y 418.225,Z 472.385,A -85,B 0,C 180,E1 -10237.263,E2 -10237.263} C_VEL
LIN {X 0,Y 418.27,Z 472.386,A -85,B 0,C 180,E1 -10240.363,E2 -10240.363} C_VEL
LIN {X 0,Y 418.304,Z 472.375,A -85,B 0,C 180,E1 -10243.404,E2 -10243.404} C_VEL
LIN {X 0,Y 418.333,Z 472.373,A -85,B 0,C 180,E1 -10246.998,E2 -10246.998} C_VEL
LIN {X 0,Y 418.328,Z 472.378,A -85,B 0,C 180,E1 -10250.328,E2 -10250.328} C_VEL
LIN {X 0,Y 418.499,Z 472.355,A -85,B 0,C 180,E1 -10252.279,E2 -10252.279} C_VEL
LIN {X 0,Y 418.493,Z 472.355,A -85,B 0,C 180,E1 -10254.217,E2 -10254.217} C_VEL
LIN {X 0,Y 418.529,Z 472.349,A -85,B 0,C 180,E1 -10258.075,E2 -10258.075} C_VEL
LIN {X 0,Y 418.657,Z 472.332,A -85,B 0,C 180,E1 -10260,E2 -10260} C_VEL
LIN {X 0,Y 418.495,Z 472.355,A -85,B 0,C 180,E1 -10262.887,E2 -10262.887} C_VEL
LIN {X 0,Y 418.476,Z 472.359,A -85,B 0,C 180,E1 -10266.751,E2 -10266.751} C_VEL
LIN {X 0,Y 418.386,Z 472.371,A -85,B 0,C 180,E1 -10268.695,E2 -10268.695} C_VEL
LIN {X 0,Y 418.303,Z 472.375,A -85,B 0,C 180,E1 -10271.631,E2 -10271.631} C_VEL
LIN {X 0,Y 418.29,Z 472.384,A -85,B 0,C 180,E1 -10274.597,E2 -10274.597} C_VEL
LIN {X 0,Y 418.274,Z 472.379,A -85,B 0,C 180,E1 -10277.604,E2 -10277.604} C_VEL
LIN {X 0,Y 418.236,Z 472.391,A -85,B 0,C 180,E1 -10280.663,E2 -10280.663} C_VEL
LIN {X 0,Y 418.274,Z 472.378,A -85,B 0,C 180,E1 -10283.782,E2 -10283.782} C_VEL
LIN {X 0,Y 418.296,Z 472.379,A -85,B 0,C 180,E1 -10287.071,E2 -10287.071} C_VEL
LIN {X 0,Y 418.231,Z 472.386,A -85,B 0,C 180,E1 -10290.273,E2 -10290.273} C_VEL
LIN {X 0,Y 418.236,Z 472.383,A -85,B 0,C 180,E1 -10293.678,E2 -10293.678} C_VEL
LIN {X 0,Y 418.233,Z 472.386,A -85,B 0,C 180,E1 -10297.224,E2 -10297.224} C_VEL
LIN {X 0,Y 418.237,Z 472.383,A -85,B 0,C 180,E1 -10299.683,E2 -10299.683} C_VEL
LIN {X 0,Y 418.22,Z 472.387,A -85,B 0,C 180,E1 -10302.323,E2 -10302.323} C_VEL
LIN {X 0,Y 418.25,Z 472.386,A -85,B 0,C 180,E1 -10305.113,E2 -10305.113} C_VEL
LIN {X 0,Y 418.282,Z 472.378,A -85,B 0,C 180,E1 -10307.775,E2 -10307.775} C_VEL
LIN {X 0,Y 418.257,Z 472.382,A -85,B 0,C 180,E1 -10311.561,E2 -10311.561} C_VEL
LIN {X 0,Y 418.25,Z 472.387,A -85,B 0,C 180,E1 -10315.16,E2 -10315.16} C_VEL
LIN {X 0,Y 418.237,Z 472.385,A -85,B 0,C 180,E1 -10317.473,E2 -10317.473} C_VEL
LIN {X 0,Y 418.26,Z 472.387,A -85,B 0,C 180,E1 -10320.897,E2 -10320.897} C_VEL
LIN {X 0,Y 418.263,Z 472.38,A -85,B 0,C 180,E1 -10324.098,E2 -10324.098} C_VEL
LIN {X 0,Y 418.232,Z 472.389,A -85,B 0,C 180,E1 -10327.265,E2 -10327.265} C_VEL
LIN {X 0,Y 418.278,Z 472.379,A -85,B 0,C 180,E1 -10330.366,E2 -10330.366} C_VEL
LIN {X 0,Y 418.312,Z 472.377,A -85,B 0,C 180,E1 -10333.406,E2 -10333.406} C_VEL
LIN {X 0,Y 418.342,Z 472.376,A -85,B 0,C 180,E1 -10337.001,E2 -10337.001} C_VEL
LIN {X 0,Y 418.338,Z 472.375,A -85,B 0,C 180,E1 -10340.33,E2 -10340.33} C_VEL
LIN {X 0,Y 418.492,Z 472.355,A -85,B 0,C 180,E1 -10343.251,E2 -10343.251} C_VEL
LIN {X 0,Y 418.339,Z 472.53,A -85,B 0,C 180,E1 -10345.648,E2 -10345.648} C_VEL
LIN {X 0,Y 418.576,Z 473.593,A -85,B 0,C 180,E1 -10345.814,E2 -10345.814} C_VEL
LIN {X 0,Y 423.397,Z 486.608,A -85,B 0,C 180,E1 -10346.244,E2 -10346.244} C_VEL
LIN {X 0,Y 422.875,Z 553.517,A -85,B 0,C 180,E1 -10347.404,E2 -10347.404} C_VEL
LIN {X 0,Y 422.812,Z 567.068,A -85,B 0,C 180,E1 -10347.837,E2 -10347.837} C_VEL
LIN {X 0,Y 422.561,Z 579.978,A -85,B 0,C 180,E1 -10348.453,E2 -10348.453} C_VEL
LIN {X 0,Y 422.31,Z 588.278,A -85,B 0,C 180,E1 -10348.973,E2 -10348.973} C_VEL
LIN {X 0,Y 421.504,Z 593.56,A -85,B 0,C 180,E1 -10349.331,E2 -10349.331} C_VEL
LIN {X 0,Y 418.302,Z 601.934,A -85,B 0,C 180,E1 -10349.921,E2 -10349.921} C_VEL
LIN {X 0,Y 415.044,Z 609.895,A -85,B 0,C 180,E1 -10350.599,E2 -10350.599} C_VEL
LIN {X 0,Y 414.14,Z 614.45,A -85,B 0,C 180,E1 -10351.09,E2 -10351.09} C_VEL
LIN {X 0,Y 413.685,Z 622.838,A -85,B 0,C 180,E1 -10352.192,E2 -10352.192} C_VEL
LIN {X 0,Y 413.112,Z 630.577,A -85,B 0,C 180,E1 -10353.415,E2 -10353.415} C_VEL
LIN {X 0,Y 412.595,Z 638.122,A -85,B 0,C 180,E1 -10354.887,E2 -10354.887} C_VEL
LIN {X 0,Y 412.199,Z 644.189,A -85,B 0,C 180,E1 -10356.364,E2 -10356.364} C_VEL
LIN {X 0,Y 411.771,Z 649.867,A -85,B 0,C 180,E1 -10358.141,E2 -10358.141} C_VEL
LIN {X 0,Y 411.462,Z 653.786,A -85,B 0,C 180,E1 -10359.836,E2 -10359.836} C_VEL
LIN {X 0,Y 411.321,Z 655.476,A -85,B 0,C 180,E1 -10360.835,E2 -10360.835} C_VEL
LIN {X 0,Y 411.231,Z 656.764,A -85,B 0,C 180,E1 -10361.836,E2 -10361.836} C_VEL
LIN {X 0,Y 411.239,Z 657.753,A -85,B 0,C 180,E1 -10363.065,E2 -10363.065} C_VEL
LIN {X 0,Y 411.264,Z 658.122,A -85,B 0,C 180,E1 -10364.854,E2 -10364.854} C_VEL
LIN {X 0,Y 411.321,Z 657.781,A -85,B 0,C 180,E1 -10365.867,E2 -10365.867} C_VEL
LIN {X 0,Y 411.454,Z 656.914,A -85,B 0,C 180,E1 -10366.957,E2 -10366.957} C_VEL
LIN {X 0,Y 411.791,Z 654.135,A -85,B 0,C 180,E1 -10368.923,E2 -10368.923} C_VEL
LIN {X 0,Y 412.151,Z 651.143,A -85,B 0,C 180,E1 -10370.306,E2 -10370.306} C_VEL
LIN {X 0,Y 412.703,Z 646.238,A -85,B 0,C 180,E1 -10372.004,E2 -10372.004} C_VEL
LIN {X 0,Y 413.298,Z 640.348,A -85,B 0,C 180,E1 -10373.553,E2 -10373.553} C_VEL
LIN {X 0,Y 414.046,Z 632.839,A -85,B 0,C 180,E1 -10375.111,E2 -10375.111} C_VEL
LIN {X 0,Y 414.766,Z 625.075,A -85,B 0,C 180,E1 -10376.412,E2 -10376.412} C_VEL
LIN {X 0,Y 415.598,Z 615.479,A -85,B 0,C 180,E1 -10377.714,E2 -10377.714} C_VEL
LIN {X 0,Y 416.306,Z 605.128,A -85,B 0,C 180,E1 -10378.842,E2 -10378.842} C_VEL
LIN {X 0,Y 417.026,Z 593.91,A -85,B 0,C 180,E1 -10379.813,E2 -10379.813} C_VEL
LIN {X 0,Y 417.515,Z 582.189,A -85,B 0,C 180,E1 -10380.604,E2 -10380.604} C_VEL
LIN {X 0,Y 417.834,Z 569.204,A -85,B 0,C 180,E1 -10381.248,E2 -10381.248} C_VEL
LIN {X 0,Y 417.977,Z 556.086,A -85,B 0,C 180,E1 -10381.684,E2 -10381.684} C_VEL
LIN {X 0,Y 418.279,Z 515.925,A -85,B 0,C 180,E1 -10382.422,E2 -10382.422} C_VEL
LIN {X 0,Y 418.629,Z 490.856,A -85,B 0,C 180,E1 -10382.863,E2 -10382.863} C_VEL
LIN {X 0,Y 411.422,Z 474.267,A -85,B 0,C 180,E1 -10383.621,E2 -10383.621} C_VEL
LIN {X 0,Y 411.235,Z 473.361,A -85,B 0,C 180,E1 -10383.814,E2 -10383.814} C_VEL
LIN {X 0,Y 411.193,Z 473.263,A -85,B 0,C 180,E1 -10386.743,E2 -10386.743} C_VEL
LIN {X 0,Y 411.213,Z 473.256,A -85,B 0,C 180,E1 -10389.728,E2 -10389.728} C_VEL
LIN {X 0,Y 411.177,Z 473.263,A -85,B 0,C 180,E1 -10393.135,E2 -10393.135} C_VEL
LIN {X 0,Y 411.173,Z 473.267,A -85,B 0,C 180,E1 -10395.882,E2 -10395.882} C_VEL
LIN {X 0,Y 411.238,Z 473.423,A -85,B 0,C 180,E1 -10399.542,E2 -10399.542} C_VEL
LIN {X 0,Y 413.924,Z 486.062,A -85,B 0,C 180,E1 -10401.914,E2 -10401.914} C_VEL
LIN {X 0,Y 414.869,Z 490.717,A -85,B 0,C 180,E1 -10402.77,E2 -10402.77} C_VEL
LIN {X 0,Y 414.215,Z 509.336,A -85,B 0,C 180,E1 -10405.951,E2 -10405.951} C_VEL
LIN {X 0,Y 413.767,Z 521.267,A -85,B 0,C 180,E1 -10407.959,E2 -10407.959} C_VEL
LIN {X 0,Y 416.019,Z 534.945,A -85,B 0,C 180,E1 -10408.367,E2 -10408.367} C_VEL
LIN {X 0,Y 416.761,Z 539.143,A -85,B 0,C 180,E1 -10408.483,E2 -10408.483} C_VEL
LIN {X 0,Y 415.191,Z 631.789,A -85,B 0,C 180,E1 -10410.323,E2 -10410.323} C_VEL
LIN {X 0,Y 414.803,Z 644.97,A -85,B 0,C 180,E1 -10410.78,E2 -10410.78} C_VEL
LIN {X 0,Y 414.265,Z 657.812,A -85,B 0,C 180,E1 -10411.432,E2 -10411.432} C_VEL
LIN {X 0,Y 413.73,Z 670.39,A -85,B 0,C 180,E1 -10412.294,E2 -10412.294} C_VEL
LIN {X 0,Y 413.028,Z 682.142,A -85,B 0,C 180,E1 -10413.334,E2 -10413.334} C_VEL
LIN {X 0,Y 412.362,Z 692.621,A -85,B 0,C 180,E1 -10414.498,E2 -10414.498} C_VEL
LIN {X 0,Y 411.734,Z 702.18,A -85,B 0,C 180,E1 -10415.817,E2 -10415.817} C_VEL
LIN {X 0,Y 411.269,Z 710.161,A -85,B 0,C 180,E1 -10417.169,E2 -10417.169} C_VEL
LIN {X 0,Y 410.808,Z 717.345,A -85,B 0,C 180,E1 -10418.683,E2 -10418.683} C_VEL
LIN {X 0,Y 410.451,Z 723.548,A -85,B 0,C 180,E1 -10420.35,E2 -10420.35} C_VEL
LIN {X 0,Y 410.232,Z 728.285,A -85,B 0,C 180,E1 -10422.039,E2 -10422.039} C_VEL
LIN {X 0,Y 410.048,Z 731.549,A -85,B 0,C 180,E1 -10423.705,E2 -10423.705} C_VEL
LIN {X 0,Y 409.935,Z 733.336,A -85,B 0,C 180,E1 -10425.099,E2 -10425.099} C_VEL
LIN {X 0,Y 409.907,Z 734.085,A -85,B 0,C 180,E1 -10426.112,E2 -10426.112} C_VEL
LIN {X 0,Y 410.032,Z 734.379,A -85,B 0,C 180,E1 -10427.69,E2 -10427.69} C_VEL
LIN {X 0,Y 410.049,Z 733.712,A -85,B 0,C 180,E1 -10429.133,E2 -10429.133} C_VEL
LIN {X 0,Y 410.087,Z 732.739,A -85,B 0,C 180,E1 -10430.132,E2 -10430.132} C_VEL
LIN {X 0,Y 410.205,Z 731.305,A -85,B 0,C 180,E1 -10431.13,E2 -10431.13} C_VEL
LIN {X 0,Y 410.441,Z 728.31,A -85,B 0,C 180,E1 -10432.622,E2 -10432.622} C_VEL
LIN {X 0,Y 410.656,Z 724.25,A -85,B 0,C 180,E1 -10434.107,E2 -10434.107} C_VEL
LIN {X 0,Y 411.14,Z 717.993,A -85,B 0,C 180,E1 -10435.834,E2 -10435.834} C_VEL
LIN {X 0,Y 411.594,Z 711.146,A -85,B 0,C 180,E1 -10437.309,E2 -10437.309} C_VEL
LIN {X 0,Y 412.314,Z 702.558,A -85,B 0,C 180,E1 -10438.779,E2 -10438.779} C_VEL
LIN {X 0,Y 412.99,Z 693.786,A -85,B 0,C 180,E1 -10440,E2 -10440} C_VEL
LIN {X 0,Y 413.786,Z 682.935,A -85,B 0,C 180,E1 -10441.217,E2 -10441.217} C_VEL
LIN {X 0,Y 414.517,Z 672.139,A -85,B 0,C 180,E1 -10442.187,E2 -10442.187} C_VEL
LIN {X 0,Y 415.131,Z 661.033,A -85,B 0,C 180,E1 -10442.979,E2 -10442.979} C_VEL
LIN {X 0,Y 415.727,Z 648.264,A -85,B 0,C 180,E1 -10443.662,E2 -10443.662} C_VEL
LIN {X 0,Y 416.113,Z 636.356,A -85,B 0,C 180,E1 -10444.121,E2 -10444.121} C_VEL
LIN {X 0,Y 416.449,Z 620.556,A -85,B 0,C 180,E1 -10444.494,E2 -10444.494} C_VEL
LIN {X 0,Y 418.168,Z 539.063,A -85,B 0,C 180,E1 -10446.212,E2 -10446.212} C_VEL
LIN {X 0,Y 415.215,Z 524.676,A -85,B 0,C 180,E1 -10446.744,E2 -10446.744} C_VEL
LIN {X 0,Y 415.082,Z 523.314,A -85,B 0,C 180,E1 -10446.868,E2 -10446.868} C_VEL
LIN {X 0,Y 416.017,Z 500.433,A -85,B 0,C 180,E1 -10450.71,E2 -10450.71} C_VEL
LIN {X 0,Y 416.265,Z 494.583,A -85,B 0,C 180,E1 -10451.689,E2 -10451.689} C_VEL
LIN {X 0,Y 414.7,Z 486.23,A -85,B 0,C 180,E1 -10453.226,E2 -10453.226} C_VEL
LIN {X 0,Y 411.288,Z 473.458,A -85,B 0,C 180,E1 -10455.708,E2 -10455.708} C_VEL
LIN {X 0,Y 411.253,Z 473.259,A -85,B 0,C 180,E1 -10457.915,E2 -10457.915} C_VEL
LIN {X 0,Y 411.205,Z 473.265,A -85,B 0,C 180,E1 -10461.034,E2 -10461.034} C_VEL
LIN {X 0,Y 411.22,Z 473.262,A -85,B 0,C 180,E1 -10464.216,E2 -10464.216} C_VEL
LIN {X 0,Y 411.268,Z 473.256,A -85,B 0,C 180,E1 -10467.477,E2 -10467.477} C_VEL
LIN {X 0,Y 411.198,Z 473.266,A -85,B 0,C 180,E1 -10470.847,E2 -10470.847} C_VEL
LIN {X 0,Y 411.214,Z 473.261,A -85,B 0,C 180,E1 -10474.333,E2 -10474.333} C_VEL
LIN {X 0,Y 411.202,Z 473.262,A -85,B 0,C 180,E1 -10477.973,E2 -10477.973} C_VEL
LIN {X 0,Y 411.172,Z 473.268,A -85,B 0,C 180,E1 -10481.228,E2 -10481.228} C_VEL
LIN {X 0,Y 411.184,Z 473.265,A -85,B 0,C 180,E1 -10484.49,E2 -10484.49} C_VEL
LIN {X 0,Y 411.185,Z 473.266,A -85,B 0,C 180,E1 -10488.194,E2 -10488.194} C_VEL
LIN {X 0,Y 411.216,Z 473.248,A -85,B 0,C 180,E1 -10490.774,E2 -10490.774} C_VEL
LIN {X 0,Y 411.186,Z 473.263,A -85,B 0,C 180,E1 -10494.468,E2 -10494.468} C_VEL
LIN {X 0,Y 411.234,Z 473.474,A -85,B 0,C 180,E1 -10496.754,E2 -10496.754} C_VEL
LIN {X 0,Y 414.773,Z 487.444,A -85,B 0,C 180,E1 -10499.446,E2 -10499.446} C_VEL
LIN {X 0,Y 416.666,Z 496.742,A -85,B 0,C 180,E1 -10501.119,E2 -10501.119} C_VEL
LIN {X 0,Y 416.215,Z 504.307,A -85,B 0,C 180,E1 -10502.33,E2 -10502.33} C_VEL
LIN {X 0,Y 414.629,Z 526.025,A -85,B 0,C 180,E1 -10505.728,E2 -10505.728} C_VEL
LIN {X 0,Y 412.964,Z 551.946,A -85,B 0,C 180,E1 -10509.708,E2 -10509.708} C_VEL
LIN {X 0,Y 412.846,Z 555.146,A -85,B 0,C 180,E1 -10510.153,E2 -10510.153} C_VEL
LIN {X 0,Y 414.451,Z 568.083,A -85,B 0,C 180,E1 -10510.569,E2 -10510.569} C_VEL
LIN {X 0,Y 417.196,Z 595.303,A -85,B 0,C 180,E1 -10511.21,E2 -10511.21} C_VEL
LIN {X 0,Y 416.22,Z 666.125,A -85,B 0,C 180,E1 -10512.463,E2 -10512.463} C_VEL
LIN {X 0,Y 415.685,Z 679.466,A -85,B 0,C 180,E1 -10512.884,E2 -10512.884} C_VEL
LIN {X 0,Y 414.783,Z 692.839,A -85,B 0,C 180,E1 -10513.511,E2 -10513.511} C_VEL
LIN {X 0,Y 413.547,Z 711.343,A -85,B 0,C 180,E1 -10514.726,E2 -10514.726} C_VEL
LIN {X 0,Y 412.842,Z 722.165,A -85,B 0,C 180,E1 -10515.582,E2 -10515.582} C_VEL
LIN {X 0,Y 412.224,Z 732.789,A -85,B 0,C 180,E1 -10516.641,E2 -10516.641} C_VEL
LIN {X 0,Y 411.542,Z 741.349,A -85,B 0,C 180,E1 -10517.673,E2 -10517.673} C_VEL
LIN {X 0,Y 411.095,Z 749.806,A -85,B 0,C 180,E1 -10518.91,E2 -10518.91} C_VEL
LIN {X 0,Y 410.649,Z 758.103,A -85,B 0,C 180,E1 -10520.393,E2 -10520.393} C_VEL
LIN {X 0,Y 410.384,Z 763.711,A -85,B 0,C 180,E1 -10521.628,E2 -10521.628} C_VEL
LIN {X 0,Y 410.195,Z 769.191,A -85,B 0,C 180,E1 -10523.11,E2 -10523.11} C_VEL
LIN {X 0,Y 410.165,Z 773.429,A -85,B 0,C 180,E1 -10524.591,E2 -10524.591} C_VEL
LIN {X 0,Y 410.089,Z 776.555,A -85,B 0,C 180,E1 -10526.068,E2 -10526.068} C_VEL
LIN {X 0,Y 410.179,Z 778.043,A -85,B 0,C 180,E1 -10527.052,E2 -10527.052} C_VEL
LIN {X 0,Y 410.166,Z 779.106,A -85,B 0,C 180,E1 -10528.035,E2 -10528.035} C_VEL
LIN {X 0,Y 410.159,Z 779.751,A -85,B 0,C 180,E1 -10529.017,E2 -10529.017} C_VEL
LIN {X 0,Y 410.222,Z 779.927,A -85,B 0,C 180,E1 -10529.998,E2 -10529.998} C_VEL
LIN {X 0,Y 410.184,Z 779.668,A -85,B 0,C 180,E1 -10530.98,E2 -10530.98} C_VEL
LIN {X 0,Y 410.162,Z 778.995,A -85,B 0,C 180,E1 -10531.962,E2 -10531.962} C_VEL
LIN {X 0,Y 410.193,Z 777.874,A -85,B 0,C 180,E1 -10532.945,E2 -10532.945} C_VEL
LIN {X 0,Y 410.114,Z 775.329,A -85,B 0,C 180,E1 -10534.421,E2 -10534.421} C_VEL
LIN {X 0,Y 410.132,Z 771.7,A -85,B 0,C 180,E1 -10535.9,E2 -10535.9} C_VEL
LIN {X 0,Y 410.272,Z 766.885,A -85,B 0,C 180,E1 -10537.38,E2 -10537.38} C_VEL
LIN {X 0,Y 410.459,Z 760.733,A -85,B 0,C 180,E1 -10538.863,E2 -10538.863} C_VEL
LIN {X 0,Y 410.764,Z 753.028,A -85,B 0,C 180,E1 -10540.348,E2 -10540.348} C_VEL
LIN {X 0,Y 411.213,Z 745.104,A -85,B 0,C 180,E1 -10541.583,E2 -10541.583} C_VEL
LIN {X 0,Y 411.75,Z 736.463,A -85,B 0,C 180,E1 -10542.693,E2 -10542.693} C_VEL
LIN {X 0,Y 412.306,Z 725.873,A -85,B 0,C 180,E1 -10543.804,E2 -10543.804} C_VEL
LIN {X 0,Y 412.915,Z 714.067,A -85,B 0,C 180,E1 -10544.79,E2 -10544.79} C_VEL
LIN {X 0,Y 413.699,Z 700.478,A -85,B 0,C 180,E1 -10545.644,E2 -10545.644} C_VEL
LIN {X 0,Y 414.537,Z 685.806,A -85,B 0,C 180,E1 -10546.433,E2 -10546.433} C_VEL
LIN {X 0,Y 415.144,Z 673.089,A -85,B 0,C 180,E1 -10546.914,E2 -10546.914} C_VEL
LIN {X 0,Y 415.426,Z 659.837,A -85,B 0,C 180,E1 -10547.219,E2 -10547.219} C_VEL
LIN {X 0,Y 415.994,Z 592.287,A -85,B 0,C 180,E1 -10548.388,E2 -10548.388} C_VEL
LIN {X 0,Y 412.385,Z 556.782,A -85,B 0,C 180,E1 -10549.182,E2 -10549.182} C_VEL
LIN {X 0,Y 413.603,Z 532.894,A -85,B 0,C 180,E1 -10552.739,E2 -10552.739} C_VEL
LIN {X 0,Y 415.048,Z 508.896,A -85,B 0,C 180,E1 -10556.361,E2 -10556.361} C_VEL
LIN {X 0,Y 415.874,Z 494.901,A -85,B 0,C 180,E1 -10558.505,E2 -10558.505} C_VEL
LIN {X 0,Y 412.537,Z 479.136,A -85,B 0,C 180,E1 -10561.175,E2 -10561.175} C_VEL
LIN {X 0,Y 411.251,Z 473.376,A -85,B 0,C 180,E1 -10562.222,E2 -10562.222} C_VEL
LIN {X 0,Y 411.189,Z 473.267,A -85,B 0,C 180,E1 -10565.527,E2 -10565.527} C_VEL
LIN {X 0,Y 411.169,Z 473.264,A -85,B 0,C 180,E1 -10569.227,E2 -10569.227} C_VEL
LIN {X 0,Y 411.161,Z 473.267,A -85,B 0,C 180,E1 -10572.692,E2 -10572.692} C_VEL
LIN {X 0,Y 411.159,Z 473.268,A -85,B 0,C 180,E1 -10575.879,E2 -10575.879} C_VEL
LIN {X 0,Y 411.145,Z 473.268,A -85,B 0,C 180,E1 -10578.772,E2 -10578.772} C_VEL
LIN {X 0,Y 411.175,Z 473.267,A -85,B 0,C 180,E1 -10582.024,E2 -10582.024} C_VEL
LIN {X 0,Y 411.195,Z 473.261,A -85,B 0,C 180,E1 -10585.665,E2 -10585.665} C_VEL
LIN {X 0,Y 411.178,Z 473.263,A -85,B 0,C 180,E1 -10589.151,E2 -10589.151} C_VEL
LIN {X 0,Y 411.247,Z 473.259,A -85,B 0,C 180,E1 -10592.521,E2 -10592.521} C_VEL
LIN {X 0,Y 411.205,Z 473.26,A -85,B 0,C 180,E1 -10595.783,E2 -10595.783} C_VEL
LIN {X 0,Y 411.184,Z 473.263,A -85,B 0,C 180,E1 -10598.965,E2 -10598.965} C_VEL
LIN {X 0,Y 411.239,Z 473.258,A -85,B 0,C 180,E1 -10602.084,E2 -10602.084} C_VEL
LIN {X 0,Y 411.246,Z 473.255,A -85,B 0,C 180,E1 -10605.146,E2 -10605.146} C_VEL
LIN {X 0,Y 411.272,Z 473.255,A -85,B 0,C 180,E1 -10608.167,E2 -10608.167} C_VEL
LIN {X 0,Y 411.468,Z 473.23,A -85,B 0,C 180,E1 -10612.146,E2 -10612.146} C_VEL
LIN {X 0,Y 411.456,Z 473.231,A -85,B 0,C 180,E1 -10614.117,E2 -10614.117} C_VEL
LIN {X 0,Y 411.498,Z 473.225,A -85,B 0,C 180,E1 -10618.042,E2 -10618.042} C_VEL
LIN {X 0,Y 411.627,Z 473.208,A -85,B 0,C 180,E1 -10620,E2 -10620} C_VEL
LIN {X 0,Y 411.451,Z 473.232,A -85,B 0,C 180,E1 -10622.937,E2 -10622.937} C_VEL
LIN {X 0,Y 411.444,Z 473.234,A -85,B 0,C 180,E1 -10626.867,E2 -10626.867} C_VEL
LIN {X 0,Y 411.34,Z 473.247,A -85,B 0,C 180,E1 -10628.845,E2 -10628.845} C_VEL
LIN {X 0,Y 411.271,Z 473.251,A -85,B 0,C 180,E1 -10631.833,E2 -10631.833} C_VEL
LIN {X 0,Y 411.247,Z 473.259,A -85,B 0,C 180,E1 -10634.853,E2 -10634.853} C_VEL
LIN {X 0,Y 411.238,Z 473.255,A -85,B 0,C 180,E1 -10637.915,E2 -10637.915} C_VEL
LIN {X 0,Y 411.182,Z 473.265,A -85,B 0,C 180,E1 -10641.034,E2 -10641.034} C_VEL
LIN {X 0,Y 411.213,Z 473.26,A -85,B 0,C 180,E1 -10644.216,E2 -10644.216} C_VEL
LIN {X 0,Y 411.245,Z 473.255,A -85,B 0,C 180,E1 -10647.478,E2 -10647.478} C_VEL
LIN {X 0,Y 411.176,Z 473.269,A -85,B 0,C 180,E1 -10650.848,E2 -10650.848} C_VEL
LIN {X 0,Y 411.193,Z 473.263,A -85,B 0,C 180,E1 -10654.334,E2 -10654.334} C_VEL
LIN {X 0,Y 411.186,Z 473.262,A -85,B 0,C 180,E1 -10657.974,E2 -10657.974} C_VEL
LIN {X 0,Y 411.152,Z 473.269,A -85,B 0,C 180,E1 -10661.229,E2 -10661.229} C_VEL
LIN {X 0,Y 411.178,Z 473.265,A -85,B 0,C 180,E1 -10664.49,E2 -10664.49} C_VEL
LIN {X 0,Y 411.218,Z 473.26,A -85,B 0,C 180,E1 -10667.298,E2 -10667.298} C_VEL
LIN {X 0,Y 411.222,Z 473.263,A -85,B 0,C 180,E1 -10670.779,E2 -10670.779} C_VEL
LIN {X 0,Y 411.19,Z 473.263,A -85,B 0,C 180,E1 -10674.473,E2 -10674.473} C_VEL
LIN {X 0,Y 411.198,Z 473.266,A -85,B 0,C 180,E1 -10676.875,E2 -10676.875} C_VEL
LIN {X 0,Y 411.225,Z 473.26,A -85,B 0,C 180,E1 -10680.646,E2 -10680.646} C_VEL
LIN {X 0,Y 411.23,Z 473.257,A -85,B 0,C 180,E1 -10683.621,E2 -10683.621} C_VEL
LIN {X 0,Y 411.197,Z 473.265,A -85,B 0,C 180,E1 -10686.854,E2 -10686.854} C_VEL
LIN {X 0,Y 411.209,Z 473.259,A -85,B 0,C 180,E1 -10690.052,E2 -10690.052} C_VEL
LIN {X 0,Y 411.258,Z 473.26,A -85,B 0,C 180,E1 -10693.133,E2 -10693.133} C_VEL
LIN {X 0,Y 411.301,Z 473.252,A -85,B 0,C 180,E1 -10696.897,E2 -10696.897} C_VEL
LIN {X 0,Y 411.29,Z 473.253,A -85,B 0,C 180,E1 -10700.163,E2 -10700.163} C_VEL
LIN {X 0,Y 411.459,Z 473.231,A -85,B 0,C 180,E1 -10703.135,E2 -10703.135} C_VEL
LIN {X 0,Y 411.327,Z 473.439,A -85,B 0,C 180,E1 -10705.386,E2 -10705.386} C_VEL
LIN {X 0,Y 411.569,Z 474.504,A -85,B 0,C 180,E1 -10705.544,E2 -10705.544} C_VEL
LIN {X 0,Y 416.675,Z 488.424,A -85,B 0,C 180,E1 -10706.006,E2 -10706.006} C_VEL
LIN {X 0,Y 416.036,Z 553.914,A -85,B 0,C 180,E1 -10707.157,E2 -10707.157} C_VEL
LIN {X 0,Y 415.99,Z 566.583,A -85,B 0,C 180,E1 -10707.551,E2 -10707.551} C_VEL
LIN {X 0,Y 415.755,Z 578.915,A -85,B 0,C 180,E1 -10708.125,E2 -10708.125} C_VEL
LIN {X 0,Y 415.371,Z 591.336,A -85,B 0,C 180,E1 -10708.911,E2 -10708.911} C_VEL
LIN {X 0,Y 414.825,Z 602.975,A -85,B 0,C 180,E1 -10709.878,E2 -10709.878} C_VEL
LIN {X 0,Y 414.189,Z 613.449,A -85,B 0,C 180,E1 -10710.974,E2 -10710.974} C_VEL
LIN {X 0,Y 414.14,Z 614.45,A -85,B 0,C 180,E1 -10711.09,E2 -10711.09} C_VEL
LIN {X 0,Y 413.263,Z 618.93,A -85,B 0,C 180,E1 -10711.611,E2 -10711.611} C_VEL
LIN {X 0,Y 410.047,Z 625.938,A -85,B 0,C 180,E1 -10712.481,E2 -10712.481} C_VEL
LIN {X 0,Y 406.78,Z 632.34,A -85,B 0,C 180,E1 -10713.442,E2 -10713.442} C_VEL
LIN {X 0,Y 405.837,Z 635.869,A -85,B 0,C 180,E1 -10714.098,E2 -10714.098} C_VEL
LIN {X 0,Y 405.381,Z 642.087,A -85,B 0,C 180,E1 -10715.473,E2 -10715.473} C_VEL
LIN {X 0,Y 405.022,Z 647.554,A -85,B 0,C 180,E1 -10716.978,E2 -10716.978} C_VEL
LIN {X 0,Y 404.744,Z 651.179,A -85,B 0,C 180,E1 -10718.212,E2 -10718.212} C_VEL
LIN {X 0,Y 404.409,Z 655.123,A -85,B 0,C 180,E1 -10720.01,E2 -10720.01} C_VEL
LIN {X 0,Y 404.268,Z 656.751,A -85,B 0,C 180,E1 -10721.026,E2 -10721.026} C_VEL
LIN {X 0,Y 404.203,Z 657.965,A -85,B 0,C 180,E1 -10722.045,E2 -10722.045} C_VEL
LIN {X 0,Y 404.212,Z 658.782,A -85,B 0,C 180,E1 -10723.18,E2 -10723.18} C_VEL
LIN {X 0,Y 404.257,Z 659.088,A -85,B 0,C 180,E1 -10725.118,E2 -10725.118} C_VEL
LIN {X 0,Y 404.327,Z 658.65,A -85,B 0,C 180,E1 -10726.149,E2 -10726.149} C_VEL
LIN {X 0,Y 404.476,Z 657.771,A -85,B 0,C 180,E1 -10727.182,E2 -10727.182} C_VEL
LIN {X 0,Y 404.651,Z 656.488,A -85,B 0,C 180,E1 -10728.219,E2 -10728.219} C_VEL
LIN {X 0,Y 405.01,Z 653.703,A -85,B 0,C 180,E1 -10729.78,E2 -10729.78} C_VEL
LIN {X 0,Y 405.477,Z 649.816,A -85,B 0,C 180,E1 -10731.347,E2 -10731.347} C_VEL
LIN {X 0,Y 406.062,Z 644.693,A -85,B 0,C 180,E1 -10732.92,E2 -10732.92} C_VEL
LIN {X 0,Y 406.785,Z 638.085,A -85,B 0,C 180,E1 -10734.499,E2 -10734.499} C_VEL
LIN {X 0,Y 407.577,Z 630.551,A -85,B 0,C 180,E1 -10735.939,E2 -10735.939} C_VEL
LIN {X 0,Y 408.466,Z 621.026,A -85,B 0,C 180,E1 -10737.405,E2 -10737.405} C_VEL
LIN {X 0,Y 409.248,Z 611.271,A -85,B 0,C 180,E1 -10738.602,E2 -10738.602} C_VEL
LIN {X 0,Y 410.045,Z 600.466,A -85,B 0,C 180,E1 -10739.665,E2 -10739.665} C_VEL
LIN {X 0,Y 410.612,Z 590.256,A -85,B 0,C 180,E1 -10740.47,E2 -10740.47} C_VEL
LIN {X 0,Y 411.062,Z 579.01,A -85,B 0,C 180,E1 -10741.165,E2 -10741.165} C_VEL
LIN {X 0,Y 411.257,Z 566.568,A -85,B 0,C 180,E1 -10741.731,E2 -10741.731} C_VEL
LIN {X 0,Y 411.393,Z 553.113,A -85,B 0,C 180,E1 -10742.117,E2 -10742.117} C_VEL
LIN {X 0,Y 411.994,Z 492.362,A -85,B 0,C 180,E1 -10743.222,E2 -10743.222} C_VEL
LIN {X 0,Y 404.401,Z 475.223,A -85,B 0,C 180,E1 -10744.038,E2 -10744.038} C_VEL
LIN {X 0,Y 404.194,Z 474.245,A -85,B 0,C 180,E1 -10744.238,E2 -10744.238} C_VEL
LIN {X 0,Y 404.144,Z 474.14,A -85,B 0,C 180,E1 -10747.493,E2 -10747.493} C_VEL
LIN {X 0,Y 404.152,Z 474.137,A -85,B 0,C 180,E1 -10750.081,E2 -10750.081} C_VEL
LIN {X 0,Y 404.157,Z 474.137,A -85,B 0,C 180,E1 -10753.085,E2 -10753.085} C_VEL
LIN {X 0,Y 404.153,Z 474.142,A -85,B 0,C 180,E1 -10755.927,E2 -10755.927} C_VEL
LIN {X 0,Y 404.182,Z 474.33,A -85,B 0,C 180,E1 -10759.29,E2 -10759.29} C_VEL
LIN {X 0,Y 406.794,Z 486.198,A -85,B 0,C 180,E1 -10761.541,E2 -10761.541} C_VEL
LIN {X 0,Y 407.942,Z 492.047,A -85,B 0,C 180,E1 -10762.623,E2 -10762.623} C_VEL
LIN {X 0,Y 407.391,Z 508.677,A -85,B 0,C 180,E1 -10765.491,E2 -10765.491} C_VEL
LIN {X 0,Y 406.916,Z 521.804,A -85,B 0,C 180,E1 -10767.693,E2 -10767.693} C_VEL
LIN {X 0,Y 409.908,Z 539.911,A -85,B 0,C 180,E1 -10768.219,E2 -10768.219} C_VEL
LIN {X 0,Y 408.316,Z 631.793,A -85,B 0,C 180,E1 -10770.092,E2 -10770.092} C_VEL
LIN {X 0,Y 407.938,Z 644.323,A -85,B 0,C 180,E1 -10770.523,E2 -10770.523} C_VEL
LIN {X 0,Y 407.402,Z 656.259,A -85,B 0,C 180,E1 -10771.117,E2 -10771.117} C_VEL
LIN {X 0,Y 406.875,Z 668.025,A -85,B 0,C 180,E1 -10771.897,E2 -10771.897} C_VEL
LIN {X 0,Y 406.233,Z 679.357,A -85,B 0,C 180,E1 -10772.852,E2 -10772.852} C_VEL
LIN {X 0,Y 405.498,Z 690.536,A -85,B 0,C 180,E1 -10774.048,E2 -10774.048} C_VEL
LIN {X 0,Y 404.867,Z 700.56,A -85,B 0,C 180,E1 -10775.38,E2 -10775.38} C_VEL
LIN {X 0,Y 404.294,Z 709.431,A -85,B 0,C 180,E1 -10776.856,E2 -10776.856} C_VEL
LIN {X 0,Y 403.835,Z 716.439,A -85,B 0,C 180,E1 -10778.296,E2 -10778.296} C_VEL
LIN {X 0,Y 403.546,Z 721.649,A -85,B 0,C 180,E1 -10779.616,E2 -10779.616} C_VEL
LIN {X 0,Y 403.263,Z 726.612,A -85,B 0,C 180,E1 -10781.191,E2 -10781.191} C_VEL
LIN {X 0,Y 403.073,Z 730.291,A -85,B 0,C 180,E1 -10782.758,E2 -10782.758} C_VEL
LIN {X 0,Y 402.962,Z 732.088,A -85,B 0,C 180,E1 -10783.797,E2 -10783.797} C_VEL
LIN {X 0,Y 402.862,Z 733.449,A -85,B 0,C 180,E1 -10784.831,E2 -10784.831} C_VEL
LIN {X 0,Y 402.829,Z 734.337,A -85,B 0,C 180,E1 -10785.863,E2 -10785.863} C_VEL
LIN {X 0,Y 402.95,Z 734.805,A -85,B 0,C 180,E1 -10787.617,E2 -10787.617} C_VEL
LIN {X 0,Y 402.978,Z 734.336,A -85,B 0,C 180,E1 -10788.94,E2 -10788.94} C_VEL
LIN {X 0,Y 402.992,Z 733.455,A -85,B 0,C 180,E1 -10789.957,E2 -10789.957} C_VEL
LIN {X 0,Y 403.112,Z 732.157,A -85,B 0,C 180,E1 -10790.973,E2 -10790.973} C_VEL
LIN {X 0,Y 403.359,Z 729.35,A -85,B 0,C 180,E1 -10792.492,E2 -10792.492} C_VEL
LIN {X 0,Y 403.59,Z 725.493,A -85,B 0,C 180,E1 -10794.003,E2 -10794.003} C_VEL
LIN {X 0,Y 403.965,Z 720.448,A -85,B 0,C 180,E1 -10795.51,E2 -10795.51} C_VEL
LIN {X 0,Y 404.565,Z 712.87,A -85,B 0,C 180,E1 -10797.262,E2 -10797.262} C_VEL
LIN {X 0,Y 405.304,Z 704.654,A -85,B 0,C 180,E1 -10798.758,E2 -10798.758} C_VEL
LIN {X 0,Y 406.001,Z 696.229,A -85,B 0,C 180,E1 -10800,E2 -10800} C_VEL
LIN {X 0,Y 406.834,Z 685.918,A -85,B 0,C 180,E1 -10801.238,E2 -10801.238} C_VEL
LIN {X 0,Y 407.561,Z 675.714,A -85,B 0,C 180,E1 -10802.224,E2 -10802.224} C_VEL
LIN {X 0,Y 408.242,Z 663.854,A -85,B 0,C 180,E1 -10803.133,E2 -10803.133} C_VEL
LIN {X 0,Y 408.95,Z 651.058,A -85,B 0,C 180,E1 -10803.874,E2 -10803.874} C_VEL
LIN {X 0,Y 409.398,Z 637.976,A -85,B 0,C 180,E1 -10804.411,E2 -10804.411} C_VEL
LIN {X 0,Y 409.719,Z 623.442,A -85,B 0,C 180,E1 -10804.784,E2 -10804.784} C_VEL
LIN {X 0,Y 411.759,Z 540.98,A -85,B 0,C 180,E1 -10806.568,E2 -10806.568} C_VEL
LIN {X 0,Y 409.215,Z 527.833,A -85,B 0,C 180,E1 -10807.056,E2 -10807.056} C_VEL
LIN {X 0,Y 408.441,Z 524.244,A -85,B 0,C 180,E1 -10807.229,E2 -10807.229} C_VEL
LIN {X 0,Y 409.362,Z 502.638,A -85,B 0,C 180,E1 -10810.886,E2 -10810.886} C_VEL
LIN {X 0,Y 409.485,Z 495.417,A -85,B 0,C 180,E1 -10812.112,E2 -10812.112} C_VEL
LIN {X 0,Y 407.732,Z 486.993,A -85,B 0,C 180,E1 -10813.71,E2 -10813.71} C_VEL
LIN {X 0,Y 404.746,Z 476.067,A -85,B 0,C 180,E1 -10815.872,E2 -10815.872} C_VEL
LIN {X 0,Y 404.236,Z 474.233,A -85,B 0,C 180,E1 -10816.312,E2 -10816.312} C_VEL
LIN {X 0,Y 404.171,Z 474.143,A -85,B 0,C 180,E1 -10819.293,E2 -10819.293} C_VEL
LIN {X 0,Y 404.159,Z 474.144,A -85,B 0,C 180,E1 -10822.832,E2 -10822.832} C_VEL
LIN {X 0,Y 404.19,Z 474.138,A -85,B 0,C 180,E1 -10825.766,E2 -10825.766} C_VEL
LIN {X 0,Y 404.204,Z 474.135,A -85,B 0,C 180,E1 -10827.999,E2 -10827.999} C_VEL
LIN {X 0,Y 404.148,Z 474.141,A -85,B 0,C 180,E1 -10831.558,E2 -10831.558} C_VEL
LIN {X 0,Y 404.193,Z 474.138,A -85,B 0,C 180,E1 -10835.016,E2 -10835.016} C_VEL
LIN {X 0,Y 404.161,Z 474.142,A -85,B 0,C 180,E1 -10838.757,E2 -10838.757} C_VEL
LIN {X 0,Y 404.131,Z 474.144,A -85,B 0,C 180,E1 -10841.599,E2 -10841.599} C_VEL
LIN {X 0,Y 404.154,Z 474.141,A -85,B 0,C 180,E1 -10844.521,E2 -10844.521} C_VEL
LIN {X 0,Y 404.145,Z 474.143,A -85,B 0,C 180,E1 -10847.295,E2 -10847.295} C_VEL
LIN {X 0,Y 404.177,Z 474.137,A -85,B 0,C 180,E1 -10849.955,E2 -10849.955} C_VEL
LIN {X 0,Y 404.142,Z 474.133,A -85,B 0,C 180,E1 -10853.125,E2 -10853.125} C_VEL
LIN {X 0,Y 404.2,Z 474.266,A -85,B 0,C 180,E1 -10856.312,E2 -10856.312} C_VEL
LIN {X 0,Y 407.663,Z 487.979,A -85,B 0,C 180,E1 -10859.04,E2 -10859.04} C_VEL
LIN {X 0,Y 409.874,Z 498.54,A -85,B 0,C 180,E1 -10860.985,E2 -10860.985} C_VEL
LIN {X 0,Y 408.863,Z 512.248,A -85,B 0,C 180,E1 -10863.205,E2 -10863.205} C_VEL
LIN {X 0,Y 407.098,Z 535.406,A -85,B 0,C 180,E1 -10866.873,E2 -10866.873} C_VEL
LIN {X 0,Y 405.973,Z 553.14,A -85,B 0,C 180,E1 -10869.621,E2 -10869.621} C_VEL
LIN {X 0,Y 406.649,Z 558.49,A -85,B 0,C 180,E1 -10869.859,E2 -10869.859} C_VEL
LIN {X 0,Y 408.823,Z 577.257,A -85,B 0,C 180,E1 -10870.434,E2 -10870.434} C_VEL
LIN {X 0,Y 410.545,Z 595.758,A -85,B 0,C 180,E1 -10870.871,E2 -10870.871} C_VEL
LIN {X 0,Y 409.507,Z 665.622,A -85,B 0,C 180,E1 -10872.134,E2 -10872.134} C_VEL
LIN {X 0,Y 408.953,Z 678.763,A -85,B 0,C 180,E1 -10872.561,E2 -10872.561} C_VEL
LIN {X 0,Y 408.072,Z 691.472,A -85,B 0,C 180,E1 -10873.167,E2 -10873.167} C_VEL
LIN {X 0,Y 406.703,Z 711.5,A -85,B 0,C 180,E1 -10874.462,E2 -10874.462} C_VEL
LIN {X 0,Y 405.85,Z 723.449,A -85,B 0,C 180,E1 -10875.456,E2 -10875.456} C_VEL
LIN {X 0,Y 405.16,Z 734.377,A -85,B 0,C 180,E1 -10876.607,E2 -10876.607} C_VEL
LIN {X 0,Y 404.47,Z 742.97,A -85,B 0,C 180,E1 -10877.709,E2 -10877.709} C_VEL
LIN {X 0,Y 403.971,Z 751.099,A -85,B 0,C 180,E1 -10878.966,E2 -10878.966} C_VEL
LIN {X 0,Y 403.555,Z 759.012,A -85,B 0,C 180,E1 -10880.475,E2 -10880.475} C_VEL
LIN {X 0,Y 403.231,Z 765.374,A -85,B 0,C 180,E1 -10881.983,E2 -10881.983} C_VEL
LIN {X 0,Y 403.064,Z 770.905,A -85,B 0,C 180,E1 -10883.659,E2 -10883.659} C_VEL
LIN {X 0,Y 403.081,Z 774.239,A -85,B 0,C 180,E1 -10884.997,E2 -10884.997} C_VEL
LIN {X 0,Y 403.004,Z 776.2,A -85,B 0,C 180,E1 -10885.998,E2 -10885.998} C_VEL
LIN {X 0,Y 403.075,Z 777.676,A -85,B 0,C 180,E1 -10887,E2 -10887} C_VEL
LIN {X 0,Y 403.089,Z 778.729,A -85,B 0,C 180,E1 -10888,E2 -10888} C_VEL
LIN {X 0,Y 403.074,Z 779.359,A -85,B 0,C 180,E1 -10888.999,E2 -10888.999} C_VEL
LIN {X 0,Y 403.161,Z 779.52,A -85,B 0,C 180,E1 -10889.998,E2 -10889.998} C_VEL
LIN {X 0,Y 403.097,Z 779.249,A -85,B 0,C 180,E1 -10890.997,E2 -10890.997} C_VEL
LIN {X 0,Y 403.086,Z 778.564,A -85,B 0,C 180,E1 -10891.997,E2 -10891.997} C_VEL
LIN {X 0,Y 403.104,Z 777.413,A -85,B 0,C 180,E1 -10892.996,E2 -10892.996} C_VEL
LIN {X 0,Y 403.041,Z 774.835,A -85,B 0,C 180,E1 -10894.499,E2 -10894.499} C_VEL
LIN {X 0,Y 403.066,Z 771.167,A -85,B 0,C 180,E1 -10896.003,E2 -10896.003} C_VEL
LIN {X 0,Y 403.188,Z 766.305,A -85,B 0,C 180,E1 -10897.51,E2 -10897.51} C_VEL
LIN {X 0,Y 403.376,Z 760.099,A -85,B 0,C 180,E1 -10899.02,E2 -10899.02} C_VEL
LIN {X 0,Y 403.731,Z 752.333,A -85,B 0,C 180,E1 -10900.53,E2 -10900.53} C_VEL
LIN {X 0,Y 404.201,Z 744.316,A -85,B 0,C 180,E1 -10901.787,E2 -10901.787} C_VEL
LIN {X 0,Y 404.703,Z 736.67,A -85,B 0,C 180,E1 -10902.79,E2 -10902.79} C_VEL
LIN {X 0,Y 405.221,Z 726.599,A -85,B 0,C 180,E1 -10903.883,E2 -10903.883} C_VEL
LIN {X 0,Y 405.898,Z 714.577,A -85,B 0,C 180,E1 -10904.923,E2 -10904.923} C_VEL
LIN {X 0,Y 406.655,Z 702.314,A -85,B 0,C 180,E1 -10905.729,E2 -10905.729} C_VEL
LIN {X 0,Y 407.726,Z 683.924,A -85,B 0,C 180,E1 -10906.715,E2 -10906.715} C_VEL
LIN {X 0,Y 408.308,Z 670.644,A -85,B 0,C 180,E1 -10907.206,E2 -10907.206} C_VEL
LIN {X 0,Y 408.598,Z 654.561,A -85,B 0,C 180,E1 -10907.548,E2 -10907.548} C_VEL
LIN {X 0,Y 409.222,Z 593.558,A -85,B 0,C 180,E1 -10908.619,E2 -10908.619} C_VEL
LIN {X 0,Y 405.41,Z 556.099,A -85,B 0,C 180,E1 -10909.459,E2 -10909.459} C_VEL
LIN {X 0,Y 405.612,Z 550.421,A -85,B 0,C 180,E1 -10910.274,E2 -10910.274} C_VEL
LIN {X 0,Y 406.924,Z 527.734,A -85,B 0,C 180,E1 -10913.742,E2 -10913.742} C_VEL
LIN {X 0,Y 408.343,Z 505.757,A -85,B 0,C 180,E1 -10917.133,E2 -10917.133} C_VEL
LIN {X 0,Y 408.938,Z 496.444,A -85,B 0,C 180,E1 -10918.583,E2 -10918.583} C_VEL
LIN {X 0,Y 406.019,Z 482.337,A -85,B 0,C 180,E1 -10921.006,E2 -10921.006} C_VEL
LIN {X 0,Y 404.188,Z 474.237,A -85,B 0,C 180,E1 -10922.495,E2 -10922.495} C_VEL
LIN {X 0,Y 404.173,Z 474.14,A -85,B 0,C 180,E1 -10925.188,E2 -10925.188} C_VEL
LIN {X 0,Y 404.125,Z 474.142,A -85,B 0,C 180,E1 -10928.758,E2 -10928.758} C_VEL
LIN {X 0,Y 404.1,Z 474.145,A -85,B 0,C 180,E1 -10931.595,E2 -10931.595} C_VEL
LIN {X 0,Y 404.135,Z 474.143,A -85,B 0,C 180,E1 -10934.52,E2 -10934.52} C_VEL
LIN {X 0,Y 404.122,Z 474.141,A -85,B 0,C 180,E1 -10937.293,E2 -10937.293} C_VEL
LIN {X 0,Y 404.122,Z 474.145,A -85,B 0,C 180,E1 -10939.949,E2 -10939.949} C_VEL
LIN {X 0,Y 404.124,Z 474.141,A -85,B 0,C 180,E1 -10943.124,E2 -10943.124} C_VEL
LIN {X 0,Y 404.134,Z 474.146,A -85,B 0,C 180,E1 -10946.186,E2 -10946.186} C_VEL
LIN {X 0,Y 404.134,Z 474.141,A -85,B 0,C 180,E1 -10949.714,E2 -10949.714} C_VEL
LIN {X 0,Y 404.181,Z 474.134,A -85,B 0,C 180,E1 -10953.121,E2 -10953.121} C_VEL
LIN {X 0,Y 404.16,Z 474.137,A -85,B 0,C 180,E1 -10955.333,E2 -10955.333} C_VEL
LIN {X 0,Y 404.147,Z 474.143,A -85,B 0,C 180,E1 -10958.581,E2 -10958.581} C_VEL
LIN {X 0,Y 404.196,Z 474.133,A -85,B 0,C 180,E1 -10961.761,E2 -10961.761} C_VEL
LIN {X 0,Y 404.192,Z 474.135,A -85,B 0,C 180,E1 -10964.881,E2 -10964.881} C_VEL
LIN {X 0,Y 404.244,Z 474.128,A -85,B 0,C 180,E1 -10967.958,E2 -10967.958} C_VEL
LIN {X 0,Y 404.419,Z 474.107,A -85,B 0,C 180,E1 -10972.099,E2 -10972.099} C_VEL
LIN {X 0,Y 404.405,Z 474.108,A -85,B 0,C 180,E1 -10974.014,E2 -10974.014} C_VEL
LIN {X 0,Y 404.467,Z 474.1,A -85,B 0,C 180,E1 -10978.008,E2 -10978.008} C_VEL
LIN {X 0,Y 404.596,Z 474.084,A -85,B 0,C 180,E1 -10980,E2 -10980} C_VEL
LIN {X 0,Y 404.408,Z 474.108,A -85,B 0,C 180,E1 -10982.988,E2 -10982.988} C_VEL
LIN {X 0,Y 404.395,Z 474.11,A -85,B 0,C 180,E1 -10986.987,E2 -10986.987} C_VEL
LIN {X 0,Y 404.245,Z 474.127,A -85,B 0,C 180,E1 -10990.012,E2 -10990.012} C_VEL
LIN {X 0,Y 404.252,Z 474.127,A -85,B 0,C 180,E1 -10993.211,E2 -10993.211} C_VEL
LIN {X 0,Y 404.201,Z 474.135,A -85,B 0,C 180,E1 -10997.007,E2 -10997.007} C_VEL
LIN {X 0,Y 404.149,Z 474.141,A -85,B 0,C 180,E1 -11000.352,E2 -11000.352} C_VEL
LIN {X 0,Y 404.155,Z 474.137,A -85,B 0,C 180,E1 -11003.575,E2 -11003.575} C_VEL
LIN {X 0,Y 404.17,Z 474.135,A -85,B 0,C 180,E1 -11005.767,E2 -11005.767} C_VEL
LIN {X 0,Y 404.182,Z 474.134,A -85,B 0,C 180,E1 -11008,E2 -11008} C_VEL
LIN {X 0,Y 404.126,Z 474.141,A -85,B 0,C 180,E1 -11011.559,E2 -11011.559} C_VEL
LIN {X 0,Y 404.173,Z 474.14,A -85,B 0,C 180,E1 -11015.017,E2 -11015.017} C_VEL
LIN {X 0,Y 404.144,Z 474.145,A -85,B 0,C 180,E1 -11018.758,E2 -11018.758} C_VEL
LIN {X 0,Y 404.112,Z 474.143,A -85,B 0,C 180,E1 -11021.601,E2 -11021.601} C_VEL
LIN {X 0,Y 404.146,Z 474.142,A -85,B 0,C 180,E1 -11024.525,E2 -11024.525} C_VEL
LIN {X 0,Y 404.196,Z 474.135,A -85,B 0,C 180,E1 -11027.306,E2 -11027.306} C_VEL
LIN {X 0,Y 404.158,Z 474.137,A -85,B 0,C 180,E1 -11029.957,E2 -11029.957} C_VEL
LIN {X 0,Y 404.131,Z 474.145,A -85,B 0,C 180,E1 -11033.125,E2 -11033.125} C_VEL
LIN {X 0,Y 404.136,Z 474.14,A -85,B 0,C 180,E1 -11036.189,E2 -11036.189} C_VEL
LIN {X 0,Y 404.137,Z 474.14,A -85,B 0,C 180,E1 -11039.716,E2 -11039.716} C_VEL
LIN {X 0,Y 404.188,Z 474.139,A -85,B 0,C 180,E1 -11043.125,E2 -11043.125} C_VEL
LIN {X 0,Y 404.17,Z 474.139,A -85,B 0,C 180,E1 -11045.336,E2 -11045.336} C_VEL
